// ============================================================
// ADD TO GVL - HMI ROBOT B
// Các biến này mirror trực tiếp biến HMI Robot A.
// AB_StepBlockClipboard / AB_StepCopyCount vẫn dùng chung để có thể copy block step.
// ============================================================
VAR_GLOBAL
    B_PointClipboardName : STRING(20);
    B_PointClipboardR : REAL;
    B_PointClipboardSourceNo : INT;
    B_PointClipboardValid : BOOL;
    B_PointClipboardX : REAL;
    B_PointClipboardY : REAL;
    B_PointClipboardZ : REAL;
    B_StepClipboard : ST_RobotStep;
    B_StepClipboardValid : BOOL;
    B_StepCopyEnd : INT;
    B_StepCopyStart : INT;
    HMI_B_ChangeSelectedPoint : BOOL;
    HMI_B_CondCmdReq : INT;
    HMI_B_CondCmd_Down : BOOL;
    HMI_B_CondCmd_GoBot : BOOL;
    HMI_B_CondCmd_GoTop : BOOL;
    HMI_B_CondCmd_PageDown : BOOL;
    HMI_B_CondCmd_PageUp : BOOL;
    HMI_B_CondCmd_Up : BOOL;
    HMI_B_CondCopied : ST_Condition;
    HMI_B_CondEditEnable : BOOL;
    HMI_B_CondEditIndex : ARRAY[0..10] OF INT;
    HMI_B_CondEditLinkNext : ARRAY[0..10] OF INT;
    HMI_B_CondEditName : STRING(20);
    HMI_B_CondEditNo : INT;
    HMI_B_CondEditNote : ARRAY[0..10] OF STRING(30);
    HMI_B_CondEditOperator : ARRAY[0..10] OF INT;
    HMI_B_CondEditRowEnable : ARRAY[0..10] OF BOOL;
    HMI_B_CondEditSetValue : ARRAY[0..10] OF DINT;
    HMI_B_CondEditSource : ARRAY[0..10] OF INT;
    HMI_B_CondMonActualValue : ARRAY[0..10] OF DINT;
    HMI_B_CondMonFinalResult : BOOL;
    HMI_B_CondMonRowResult : ARRAY[0..10] OF BOOL;
    HMI_B_CondMonitorEnable : BOOL;
    HMI_B_CondRowSelect : ARRAY[0..10] OF BOOL;
    HMI_B_CondSelectedCmd : INT;
    HMI_B_CondSelectedNo : INT;
    HMI_B_CondViewEnable : ARRAY[0..10] OF BOOL;
    HMI_B_CondViewName : ARRAY[0..10] OF STRING(20);
    HMI_B_CondViewNo : ARRAY[0..10] OF INT;
    HMI_B_CondViewResult : ARRAY[0..10] OF BOOL;
    HMI_B_CondViewStart : INT;
    HMI_B_CopyEndStep : INT;
    HMI_B_CopyStartStep : INT;
    HMI_B_EditCmd : E_RobotCmd;
    HMI_B_EditCmdReq : INT;
    HMI_B_EditCmdReq_Arr : ARRAY[0..20] OF BOOL;
    HMI_B_EditGroupCmd : INT;
    HMI_B_EditNote : STRING(20);
    HMI_B_EditP1 : INT;
    HMI_B_EditP2 : INT;
    HMI_B_EditP3 : DINT;
    HMI_B_EditP4 : INT;
    HMI_B_EditP5 : INT;
    HMI_B_EditPointReq : INT;
    HMI_B_EditPointReq_Arr : ARRAY[0..10] OF BOOL;
    HMI_B_EditSelgroupCmd : ARRAY[0..10] OF BOOL;
    HMI_B_EditStepNo : INT;
    HMI_B_Edit_PointNo : INT;
    HMI_B_Edit_Pos_Name : STRING(20);
    HMI_B_Edit_Pos_R : REAL;
    HMI_B_Edit_Pos_X : REAL;
    HMI_B_Edit_Pos_Y : REAL;
    HMI_B_Edit_Pos_Z : REAL;
    HMI_B_Edit_Trigger_Windown_Cmd : ARRAY[0..10] OF BOOL;
    HMI_B_PointNo : ARRAY[0..10] OF INT;
    HMI_B_PointNoSelected : INT;
    HMI_B_PointViewCmd : INT;
    HMI_B_RowSelect : ARRAY[0..10] OF BOOL;
    HMI_B_RowSelectedCmd : INT;
    HMI_B_RowSelectedPoint : INT;
    HMI_B_RowSelectedPoint_Array : ARRAY[0..10] OF BOOL;
    HMI_B_SelectedStepNo : INT;
    HMI_B_ViewCmd : ARRAY[0..10] OF INT;
    HMI_B_ViewCmd_Go_Bot : BOOL;
    HMI_B_ViewCmd_Go_Bot_Old : BOOL;
    HMI_B_ViewCmd_Go_Top : BOOL;
    HMI_B_ViewCmd_Go_Top_Old : BOOL;
    HMI_B_ViewCmd_Page_Down : BOOL;
    HMI_B_ViewCmd_Page_Down_Old : BOOL;
    HMI_B_ViewCmd_Page_Up : BOOL;
    HMI_B_ViewCmd_Page_Up_Old : BOOL;
    HMI_B_ViewCmd_Scroll_Down : BOOL;
    HMI_B_ViewCmd_Scroll_Down_Old : BOOL;
    HMI_B_ViewCmd_Scroll_Up : BOOL;
    HMI_B_ViewCmd_Scroll_Up_Old : BOOL;
    HMI_B_ViewGroupCmd : ARRAY[0..10] OF INT;
    HMI_B_ViewNote : ARRAY[0..10] OF STRING(20);
    HMI_B_ViewP1 : ARRAY[0..10] OF INT;
    HMI_B_ViewP2 : ARRAY[0..10] OF INT;
    HMI_B_ViewP3 : ARRAY[0..10] OF DINT;
    HMI_B_ViewP4 : ARRAY[0..10] OF INT;
    HMI_B_ViewP5 : ARRAY[0..10] OF INT;
    HMI_B_ViewP6 : ARRAY[0..10] OF INT;
    HMI_B_ViewStartPoint : INT;
    HMI_B_ViewStartStep : INT := 1;
    HMI_B_ViewStepNo : ARRAY[0..10] OF INT;
    HMI_B_View_Pos_Name : ARRAY[0..10] OF STRING(20);
    HMI_B_View_Pos_R : ARRAY[0..10] OF REAL;
    HMI_B_View_Pos_X : ARRAY[0..10] OF REAL;
    HMI_B_View_Pos_Y : ARRAY[0..10] OF REAL;
    HMI_B_View_Pos_Z : ARRAY[0..10] OF REAL;
END_VAR

//=============================================================================
// GVL: LOGICAL IO - ROBOT B
//-----------------------------------------------------------------------------
// IO vật lý nên được Map vào các mảng này tại một chương trình riêng.
//=============================================================================
VAR_GLOBAL

    // Command và Status của lệnh TRACK_ON.
	g_stMultiTrackCommandB : ST_MultiToolTrackingCommand;
	g_stMultiTrackStatusB : ST_MultiToolTrackingStatus;
	
	// Cấu hình và Runtime Tool Robot A.
	g_aToolConfigB : ARRAY[0..C_MAX_TOOLS] OF ST_ToolConfig;
	g_aToolStatusB : ARRAY[0..C_MAX_TOOLS] OF ST_ToolStatus;
	
	// Recipe và Queue Robot A.
	g_aMultiTrackRecipeB : ARRAY[0..C_MAX_TRACK_RECIPES] OF ST_MultiToolTrackingRecipe;
	g_stTrackingObjectQueueB : ST_TrackingObjectQueue;
	
	// Cấu hình các nguồn Sensor.
    g_aSensorSourceConfigB : ARRAY[0..C_MAX_SENSOR_SOURCES] OF ST_SensorObjectSourceConfig;

  	// Cấu hình Vision Tracking cho từng Camera/Channel.
	g_aVisionTrackingSourceConfigB : ARRAY[0..C_MAX_VISION_CHANNELS] OF ST_VisionTrackingSourceConfig;
	
	// Multi-object result dành riêng cho Conveyor Tracking.
	g_aVisionTrackingMultiResultB : ARRAY[0..C_MAX_VISION_CHANNELS] OF ST_VisionTrackingMultiResult;
	
	g_aVisionAlignRecipeB : ARRAY[0..C_MAX_VISION_ALIGN_RECIPES] OF ST_VisionAlignRecipe;
	g_aVisionAlignRuntimeB : ARRAY[1..C_MAX_TOOLS] OF ST_VisionAlignToolRuntime;
	g_aTrayConfigB : ARRAY[0..C_MAX_TRAYS] OF ST_TrayConfig;
	g_aTrayRuntimeB : ARRAY[0..C_MAX_TRAYS] OF ST_TrayRuntime;

	
	// Giao tiếp giữa MultiTool Controller và Tracking Core hiện tại.
	g_xMultiTrackCoreExecuteB : BOOL;
	g_xMultiTrackCoreResetB : BOOL;
	g_xMultiTrackCoreAbortB : BOOL;
	g_xMultiTrackPickerSafeB : BOOL;
	
	g_uiMultiTrackObjectIndexB : UINT;
	g_uiMultiTrackToolIDB : UINT;
	g_stMultiTrackPickOffsetB : ST_POS;
	g_rMultiTrackApproachHeightB : REAL;
	
	// Phản hồi từ Tracking Core về MultiTool Controller.
	g_xTrackingCoreAcceptedB : BOOL;
	g_xTrackingCoreBusyB : BOOL;
	g_xTrackingCoreSyncOKB : BOOL;
	g_xTrackingCorePCSInUseB : BOOL;
	g_xTrackingCoreReleasedB : BOOL;
	g_xTrackingCoreErrorB : BOOL;
	g_udiTrackingCoreErrorIDB : UDINT;
	
	// Command Tool được Controller phát ra.
	g_stToolCommandB : ST_ToolCommand;
	
	// Chọn Tool/TCP Robot B.
	g_xSelectToolExecuteB : BOOL;
	g_uiSelectToolIDB : UINT;
	g_stSelectToolTCPB : ST_POS;
	g_xSelectToolDoneB : BOOL;
	g_xSelectToolErrorB : BOOL;
	g_udiSelectToolErrorIDB : UDINT;
	
	// IO logic Tool Robot B.
	// Nếu project đã có mảng IO chung thì dùng mảng cũ và không khai báo lại.
	g_axDIB : ARRAY[0..C_MAX_DI] OF BOOL;
	g_axDORequestToolB : ARRAY[0..C_MAX_DO] OF BOOL;
	
	// Bit test commissioning. Không dùng trong Interpreter chính thức.
	g_xMultiTrackStartTestB : BOOL;
	g_xMultiTrackResetTestB : BOOL;
	g_xMultiTrackAbortTestB : BOOL;
	g_xCreateTestTrackingObjectB : BOOL;
	
	// TRUE khi cấu hình Multi-tool Robot B đã được khởi tạo.
	g_xMultiToolConfigInitializedB : BOOL := FALSE;
	
	// Bit cho phép khởi tạo lại giá trị mặc định khi commissioning.
	g_xInitializeMultiToolConfigB : BOOL := FALSE;
	
	g_xClearTrackingQueueB : BOOL;
	g_xResetTrackingObjectSourceB : BOOL;
	
	//=============================================================================
	// TRACKING APPLICATION RESULT - ROBOT B
	//=============================================================================
	g_xTrackOKB : BOOL;              // TRUE khi lệnh Tracking gần nhất Pick đủ số lượng.
	g_xTrackErrorB : BOOL;           // TRUE khi lệnh Tracking kết thúc lỗi.
	g_udiTrackErrorIDB : UDINT;      // ErrorID của lệnh Tracking gần nhất.
	g_udiTrackDoneCommandIDB : UDINT;// CommandID đã hoàn thành.
	//=============================================================================
	// TOOL COMMAND TỪ INTERPRETER - ROBOT B
	//=============================================================================
	g_stInterpreterToolCommandB : ST_ToolCommand;
	
	g_HMI_PulsePerCycle_Cr_B: REAL;
	g_HMI_PulsePerCycle_Set_B : INT;
	
	// Cho phép test Background Vision Trigger mà chưa cần chạy TRACK_PICK.
	// Production bình thường phải để FALSE.
	g_xVisionTrackingAutoTriggerTestB : BOOL := FALSE;

END_VAR

VAR_GLOBAL
	//=========================================================================

    // VISION REQUEST FROM ROBOT INTERPRETERS

    //=========================================================================

    g_stVisionAlignRequestA : ST_VISION_ALIGN_REQUEST; // Request Vision Align từ Robot A.

    g_stVisionAlignRequestB : ST_VISION_ALIGN_REQUEST; // Request Vision Align từ Robot B.
	
END_VAR

VAR_GLOBAL
	//=============================================================================
	// V5 - CHỈ BỔ SUNG CHO ROBOT B. ROBOT A GIỮ NGUYÊN.
	// Robot A tiếp tục dùng toàn bộ biến generic hiện tại:
	// g_xTrackingMotionAccepted, g_xTrackingMotionBusy, g_xTrackingMotionDone,
	// g_xTrackingMotionError, g_udiTrackingMotionErrorID, g_xTrackingMotionAbortDone,
	// g_xTrackingVacuumOutput, g_xTrackingBlowOutput.
	//=============================================================================
	
	// Tracking state riêng Robot B.
	g_stTrackingConfig_B : ST_TRACKING_CONFIG; // Cấu hình Tracking Robot B.
	g_stTrackingQueue_B : ST_TRACKING_QUEUE; // Queue Object Robot B.
	g_stTrackingRuntime_B : ST_TRACKING_RUNTIME; // Runtime Tracking Robot B.
	
	// Motion handshake riêng Robot B.
	g_xTrackingMotionAcceptedB : BOOL; // Motion Adapter B đã nhận request.
	g_xTrackingMotionBusyB : BOOL; // Motion Tracking B đang chạy.
	g_xTrackingMotionDoneB : BOOL; // Motion Tracking B hoàn thành.
	g_xTrackingMotionErrorB : BOOL; // Motion Tracking B lỗi.
	g_udiTrackingMotionErrorIDB : UDINT; // ErrorID Motion Tracking B.
	g_xTrackingMotionAbortDoneB : BOOL; // Motion B đã Abort xong.
	
	// Debug/output riêng Robot B.
	g_xTrackingVacuumOutputB : BOOL; // VacuumCommand của Tracking Manager B.
	g_xTrackingBlowOutputB : BOOL; // BlowCommand của Tracking Manager B.
	
	// Apply Tool/TCP riêng Robot B.
	g_udiRobotBToolApplyRequestB : UDINT; // RequestID đổi Tool/TCP B.
	g_udiRobotBToolAppliedRequestB : UDINT; // RequestID B đã Apply thành công.
	g_xRobotBToolApplyBusy : BOOL; // B đang Apply Tool/TCP.
	g_xRobotBToolApplyDone : BOOL; // Xung Done Apply Tool/TCP B.
	g_xRobotBToolApplyError : BOOL; // Lỗi Apply Tool/TCP B.
	g_udiRobotBToolApplyErrorID : UDINT; // ErrorID Apply Tool/TCP B.


END_VAR

VAR_GLOBAL
	//=============================================================================
	// HMI TRACKING CONFIG - ROBOT B
	// Chỉ thêm các biến B còn thiếu. Tool Editor B đã tồn tại trong project (4).
	//=============================================================================
	
	// Sensor Source B.
	g_uiHMISensorSourceIndexB : UINT := 1;
	g_stHMISensorSourceB : ST_SensorObjectSourceConfig;
	g_xHMILoadSensorSourceB : BOOL;
	g_xHMISaveSensorSourceB : BOOL;
	g_xHMILoadSensorSourceB_All : BOOL;
	g_xHMISaveSensorSourceB_All : BOOL;
	
	// Tracking Recipe B.
	g_uiHMITrackingRecipeIndexB : UINT := 1;
	g_stHMITrackingRecipeB : ST_MultiToolTrackingRecipe;
	g_xHMILoadTrackingRecipeB : BOOL;
	g_xHMISaveTrackingRecipeB : BOOL;
	g_xHMILoadTrackingRecipeB_All : BOOL;
	g_xHMISaveTrackingRecipeB_All : BOOL;
	
	// Vision Tracking Source B.
	g_uiHMIVisionSourceIndexB : UINT := 1;
	g_stHMIVisionSourceB : ST_VisionTrackingSourceConfig;
	g_xHMILoadVisionSourceB : BOOL;
	g_xHMISaveVisionSourceB : BOOL;
	g_xHMISaveAllVisionSourceB : BOOL;
	g_xHMILoadAllVisionSourceB : BOOL := FALSE;
	
	// Tracking Config B persistence.
	g_xHMITrackingConfigSaveB : BOOL;
	g_xHMITrackingConfigReadB : BOOL;
	
	// Tool Config B persistence.
	// Không dùng g_stHMITool_Config_Save_All của A vì flag hiện tại đang Save g_aToolConfigA.
	g_xHMIToolConfigSaveAllB : BOOL;
	g_xHMIToolConfigReadAllB : BOOL;
	
	//=============================================================================
	// ROBOT B - LAST VISION ALIGN RESULT
	//=============================================================================
	B_VisionHeaderOK : BOOL;                    // Header của Result cuối hợp lệ.
	B_VisionTriggerID : UDINT;                  // TriggerID cuối cùng.
	
	B_VisionX : REAL;                           // X Vision trả về.
	B_VisionY : REAL;                           // Y Vision trả về.
	B_VisionZ : REAL;                           // Z Vision trả về.
	B_VisionA : REAL;                           // Góc Vision trả về.
	B_VisionScore : REAL;                       // Score Vision.
	
END_VAR

// Just_Motion_Control_x86_64_Linux_SM_WV/Application/PRG_ROBOT/POU_MOTION
PROGRAM POU_MOTION
VAR
	// chạy điểm
	MOVP_A :MC_MoveDirectAbsolute;
	MOVP_B :MC_MoveDirectAbsolute;
	// chạy đường thẳng
	MOVL_A: MC_MoveLinearAbsolute;
	MOVL_B: MC_MoveLinearAbsolute;
	// chạy đường tròn
	MOVC_A: MC_MoveCircularAbsolute;
	MOVC_B: MC_MoveCircularAbsolute;
	
	// Biến chạy
	RBA_BufferMode, TestA_BF_Mode: SM3_Robotics.MC_BUFFER_MODE;
	RBA_TransitionMode, TestA_Trans_Mode: SM3_Robotics.MC_TRANSITION_MODE;
	RBA_TransitionParameter, TestA_Tran_Para: ARRAY [0..(SMC_RCNST.MAX_TRANS_PARAMS - 1)] OF LREAL := [500, 0.0];
	RBA_OrientationMode, TestA_Orient_Mode: SM3_Robotics.SMC_ORIENTATION_MODE;
	RBB_BufferMode: SM3_Robotics.MC_BUFFER_MODE;
	RBB_TransitionMode: SM3_Robotics.MC_TRANSITION_MODE;
	RBB_TransitionParameter: ARRAY [0..(SMC_RCNST.MAX_TRANS_PARAMS - 1)] OF LREAL := [500, 0.0] ;
	RBB_OrientationMode: SM3_Robotics.SMC_ORIENTATION_MODE;	
	
	//RBA_MovementType: SM3_Robotics.SMC_PTP_MOVEMENT_TYPE;
	//RBb_MovementType: SM3_Robotics.SMC_PTP_MOVEMENT_TYPE;
	
	Pos_run_manual_A, Pos_run_auto_A , Pos_run_manual_B, Pos_run_auto_B ,
	Pos_Run_A, Pos_Run_A_Pre, Pos_Run_B, Pos_Run_B_Pre : SM3_Robotics.SMC_POS_REF;
	Pos_0 : SM3_Robotics.SMC_POS_REF := (c := (X:= 0,Y:= 0, Z:= 0, A:= 0, B:= 0, C:= 0));	
	MOVL_A_2: MC_MoveLinearAbsolute;
	MOVL_A_3: MC_MoveLinearAbsolute;
	MOVL_B_2: MC_MoveLinearAbsolute;
	MOVL_B_3: MC_MoveLinearAbsolute;
END_VAR

VAR // Act_go_Manual
	Excute_Run_goHome_A , AP_Man_Z_Wait_Go, AP_Man_R_Wait_Go, AP_Man_XY_Wait_Go,
	Excute_Run_goHome_B, Excute_Run_goZ_Wait_B, Excute_Run_goR_Wait_B,Excute_Run_goXY_Wait_B : BOOL;
	AP_Man_Pos_Go , Excute_Run_goPos_A_UpZ, excute_run_L_Upz_A , AP_Man_UP_Z_Go, AP_Man_Pos_Go_L,
 	Excute_Run_goPos_B, Excute_Run_goPos_B_UpZ, excute_run_L_Upz_B , excute_run_P_Upz_B, Excute_Run_goPos_B_L : BOOL;
	Excute_Run_goPos_A_UpZ_XY_BF_R, Excute_Run_goPos_A_UpZ_R_BF_XY, Excute_Run_goPos_B_UpZ_XY_BF_R, Excute_Run_goPos_B_UpZ_R_BF_XY : BOOL;
	excute_run_cam_B, excute_run_cam_A, excute_run_P_cam_B, excute_run_P_cam_A, run_calib_P_Cam_A, run_calib_P_Cam_B : BOOL;
	mode_Run_GoPosA_manual, mode_Run_GoPosB_manual: INT := 0;
	Pro_B_cam : INT;
	Running_B_Cam : BOOL;
	
	
	Other_PosA, Other_PosB: BOOL;
	PRO_A : ARRAY[0..50] OF INT;
	RuningPosA : ARRAY[0..50] OF BOOL;
	PRO_B : ARRAY[0..50] OF INT;
	RuningPosB : ARRAY[0..50] OF BOOL;
	
	T_MC1_4, T_MC2_4, Project_4_Delay_B, Project_4_Delay_A, on_Cam : TON;	
	Project_4_Delay_B1, Project_4_Delay_B2, Project_4_Delay_B3, Project_4_Delay_B4, ton_centering,  
	Project_4_Delay_A1, Project_4_Delay_A2, Project_4_Delay_A3, Project_4_Delay_A4, Project_4_Delay_A5, Project_4_Delay_A6, Project_4_Delay_A7, Project_4_Delay_A8  : TON;
	Ton_OK_MC1_4, Ton_OK_MC2_4, Ton_Limit_Test_TS, Ton_Limit_Test_VS : TON;
	Ton_tacktime, T_Delay_RB_A_Tool_1, T_Delay_RB_A_Tool_2, T_Delay_RB_B_Tool_1, T_Delay_RB_B_Tool_2 : TON;
	on_centering : WORD;
	change_fac_vel_A, change_fac_vel_B : BOOL := FALSE;
	change_fac_vel_max_A, change_fac_vel_max_A_test : BOOL := FALSE;
	change_fac_vel_max_B : BOOL := FALSE;
END_VAR

VAR // Act_go_Auto
	LOG_, LOG_A, LOG_B : FB_Write_Log(); // log file
	i_log, i_log_BF, i_log_HMI : INT;
	{region "1.Project 1"}
		Pallets_get_A,Pallets_put_A,			 
		Pallets_get_B, Pallets_put_B : FB_PALLETS;
			 
		status_MC :INT;	 
			 
		Process_1_A,Process_1_B,
		Process_2_A,Process_2_B: INT;
		Process_2_A_to_B , Process_2_B_to_A : 	 BOOL;
			 
		Process_2_A_1, Process_2_A_2, Process_2_A_3, Process_2_A_4 , 
		Process_2_B_1, Process_2_B_2, Process_2_B_3, Process_2_B_4 : BOOL;

	 
		Blink_Stop, Blink_Start : Blink_Bit; // nháy 
			 
		SR_MC : SR;
		RUN_PROJECT : BOOL;
		INIT_RUN_PROJECT : BOOL;
		AP_Auto_Pos_Go , EXCUTE_RUN_P_AUTO_B , EXCUTE_RUN_L_AUTO_A , EXCUTE_RUN_L_AUTO_B : BOOL;
			 
		Project_2_Delay, Project_2_Delay2 : TON;	  
		
		pr2_mode_A_Pick_to_B_Pick, pr2_mode_A_Pick_to_B_Place : BOOL;			 
		Move_RB_A, Move_RB_B : FB_Run_Point;
		Move_Point_Para_A, Move_Point_Para_B : Move_Point;
	{endregion}
		 
	{region "3.Project 3"}	
 
	Process_3_A,Process_3_B: INT;
	Test_Pick, Test_Place : INT;	 
	run_P_cam_B_test_pick, run_P_cam_B_test_place	: BOOL;	  
		 
	Project_3_Delay_A, Project_3_Delay_B  : TON ;
		 
	A3_Run_P, A3_Run_L, B3_Run_P, B3_Run_L : BOOL;	
	

	A_Comp, B_Comp ,Ena3, B_Allow_NextStep, A_Allow_NextStep, A_Comp_Man, B_Comp_Man, A_FB_Comp, B_FB_Comp, A_Ready, B_Ready : BOOL;
	Pro_A3, Pro_B3 : WORD; 
		  
	nextstepRtrigB, nextstepRtrigA : R_TRIG;
	// Trigger_Cmd, Trigger_Busy, Trigger_Done : BOOL;
	T1_A, T2_A : WORD;
	
	
	DATA_A_T1 , DATA_B_T1, DATA_B_T2 : WORD := 0; // 0 : NONE, 1:barcode // 2 OK 	 // 3 NG 
	DATA_MC1, Data_MC2 : WORD; // 0 NONE, 1 BUSY, 2 ALLOW PLACE, 3 ALLOW PICK 
	ALLOW_PICK_CNV, ALLOW_PLACE_CNV_OK, ALLOW_PLACE_CNV_NG_TS, ALLOW_PLACE_CNV_NG_VS  : BOOL := true;
	Pro_MC1, Pro_MC2 : WORD := 0;
	PRO_A3_,PRO_B3_  : ARRAY[0..10] OF WORD;
		 
	Wait_A3_Run , Pick_A3_Run, Place_A3_Run, Barcode_A3_Run : BOOL := FALSE;	
	 Wait_A3_Finish , Pick_A3_Finish, Place_A3_Finish, Barcode_A3_Finish : BOOL := FALSE;	
 	Allow_MC1, Allow_MC2 : BOOL;
	T_MC1, T_MC2 : TON;	 
	Wait_B3_Run , Pick_B3_T1_Run, Place_OK_B3_T1_Run, Place_NG_B3_T1_Run , Pick_B3_T2_Run , Place_Ok_B3_T2_Run , Place_NG_B3_T2_Run, Barcode_B3_Run: BOOL := FALSE;
	 Wait_B3_Finish , Pick_B3_T1_Finish, Place_OK_B3_T1_Finish, Place_NG_B3_T1_Finish , Pick_B3_T2_Finish , Place_Ok_B3_T2_Finish , Place_NG_B3_T2_Finish , Barcode_B3_Finish : BOOL := FALSE;		   
	{endregion}
    {region "4.Project 4"}
	Pro_B4, Pro_A4, Pro_A4_BF, Pro_B4_BF : WORD; 
	Ena4, Ena_Test : BOOL;	  
	nextstepRtrigB_4, nextstepRtrigA_4 : R_TRIG;
	Trigger_Cmd_4, Trigger_Busy_4, Trigger_Done_4 : BOOL;
	T1_A_4, T2_A_4 : WORD;
	R_Trig_TriggerDone_4 : R_TRIG;
	
	A4_Run_P, A4_Run_L, B4_Run_P, B4_Run_L : BOOL;	
		 
	//GVL.Pro4_.Process.DATA_TOOL_B1_IN , GVL.Pro4_.Process.DATA_TOOL_A1_IN, GVL.Pro4_.Process.DATA_TOOL_A2_OUT, GVL.Pro4_.Process.DATA_TOOL_A1_IN_OLD  : WORD := 0; // 0 : NONE, 1:barcode // 2 OK 	 // 3 NG // 4 - NG TS
	//GVL.Pro4_.Process.DATA_MC_TS, GVL.Pro4_.Process.DATA_MC_VS : WORD; // 0 NONE, 1 BUSY, 2 ALLOW PLACE, 3 ALLOW PICK OK, 4 ALLOW PICK NG, 5 ALLOW PICK NG TS
	ALLOW_PLACE_CNV_OK_4, ALLOW_PLACE_CNV_NG_TS_4, ALLOW_PLACE_CNV_NG_VS_4  : BOOL := TRUE;
	ALLOW_PICK_CNV_4 : BOOL := FALSE;	 
	Pro_MC1_4, Pro_MC2_4 : WORD := 0;
	PRO_B4_,PRO_A4_  : ARRAY[0..10] OF WORD;
		 
	Wait_B4_Run , Pick_B4_Run, Place_B4_Run, Barcode_B4_Run, Trigger_B4_Run : BOOL := FALSE;	
	 Wait_B4_Finish , Pick_B4_Finish, Place_B4_Finish, Barcode_B4_Finish, Trigger_B4_Finish : BOOL := FALSE;	
 	Allow_MC1_4, Allow_MC2_4 : BOOL;
	Ton_Test_B, Ton_Test_A: TON;	 
	delta_position_cor : REAL; 
		 
	Wait_A4_Run , Pick_A4_T1_Run, Place_OK_A4_T1_Run, Place_NG_A4_T1_Run , Pick_A4_T2_Run , Place_Ok_A4_T2_Run , Place_NG_A4_T2_Run, Place_NG_TS_A4_T2_Run, Barcode_A4_Run: BOOL := FALSE;
	 Wait_A4_Finish , Pick_A4_T1_Finish, Place_OK_A4_T1_Finish, Place_NG_A4_T1_Finish , Pick_A4_T2_Finish , Place_Ok_A4_T2_Finish , Place_NG_A4_T2_Finish ,Place_NG_TS_A4_T2_Finish, Barcode_A4_Finish : BOOL := FALSE;
	A_Test_Motion_Run, A_Test_Motion_Finish, B_Test_Motion_Run, B_Test_Motion_Finish, Just_Start_Test : BOOL;
    Process_A_Test, Process_B_Test : WORD;
		 
	D_Barcode_Ts, count_Ts, D_Barcode_Vs, count_Vs, D_Vision_Align_Ts, count_Vs_Align,
	D_CV_NG : WORD;
	T_distance_NG : TON;
	Nb_NG_VS_Cur, Nb_NG_TS_Cur : INT;
	T_Wait_Input_YL, Alarm_Barcode_VS, Alarm_Barcode_TS, Alarm_Full_NG_CONV, T_Wait_Trigger_Bar_TS, T_Wait_Trigger_Bar_VS : TON;
	HeavyAlarm, LightAlarm : BOOL;
	i_Vs_Align, i_Vs_Align_old: INT;
	Process_auto_calib: WORD;
	Run_One_Pos_Calib, Calib_first_bit, NextStep_Test, NextStep_Test_1: BOOL;
	T_Delay_Trigger_Calib: TON;
	Real_to_Word_Pos_Calib : FB_Real_TO_Word_;
	Off_Calib_FtrigB, Off_Calib_FtrigA : F_TRIG;
	Trigger_Calib_Done, Trigger_Auto_Done : R_TRIG;
	Run_Calib_VS_RB : ARRAY[0..GVL.C_MAX_VISION_CHANNELS] OF FB_CalibRunPoints;
	Trigger_VS_FB : ARRAY[0..GVL.C_MAX_VISION_CHANNELS] OF FB_TriggerVS;
	{endregion}
END_VAR

VAR
    step  : ST_RobotStep;
    bCond : BOOL;
END_VAR
//PRG_A_MotionQueueBuilder
VAR
//     step_PRG_A_MotionQueueBuilder : ST_RobotStep;
//     item_PRG_A_MotionQueueBuilder : ST_MotionQueueItem;
//     fbPush : FB_MotionQueuePush;
// 	PushReq : BOOL;
	step_PRG_A_Interpreter : ST_RobotStep;
    fbPushMotion           : FB_MotionQueuePush;
    tRunDelay              : TON;
	WhileReturnStep      : INT;
    MotionCycleResetScan : INT := 0;
END_VAR
// PRG_A_MotionManager
VAR
    fbPop : FB_MotionQueuePop;
	PopReq : BOOL;
    item_PRG_A_MotionManager  : ST_MotionQueueItem;
	freeSlot : INT;
    i : INT;
	fbMoveP : ARRAY[0..3] OF FB_RunMoveP;
    fbMoveL : ARRAY[0..3] OF FB_RunMoveL;
    fbMoveC : ARRAY[0..3] OF FB_RunMoveC;
	SlotPos : ARRAY[0..3] OF SMC_POS_REF;
    SlotMidPos : ARRAY[0..3] OF SMC_POS_REF;
    SlotEndPos : ARRAY[0..3] OF SMC_POS_REF;
	ActiveCountCalc : INT;
	WaitAcceptSlot : INT := 0;
	udiTrackCommandIDA : UDINT; // Id TrackCommand dang thuc hien
	// CommandID của TOOL_RELEASE hiện tại.
	udiToolReleaseCommandIDA : UDINT;
	
	//=============================================================================
	// VISION ALIGN
	//=============================================================================
// 	fbVisionAlignA : FB_VisionAlign;            // FB Vision Align của Robot A.
// 	xVisionAlignStartA : BOOL;                  // Start một chu trình Vision Align.
	uiVisionCameraIDA : UINT := 1;              // Camera của command hiện tại.
	uiVisionJobIDA : UINT := 1;                 // Job của command hiện tại.
	iVisionResultVarA : INT;
	xVisionStepActiveA : BOOL := FALSE;    // THÊM - ownership command Vision riêng Robot A.
	iVisionErrorIDA : INT := 0;    // Lưu ErrorID thực tế của Vision để chẩn đoán lỗi.
END_VAR
VAR
	step_PRG_B_Interpreter : ST_RobotStep;
    fbPushMotion_B           : FB_MotionQueuePush_B;
    tRunDelay_B              : TON;
	WhileReturnStep_B      : INT;
    MotionCycleResetScan_B : INT := 0;
	
	fbPop_B : FB_MotionQueuePop_B;
	PopReq_B : BOOL;
    item_PRG_B_MotionManager  : ST_MotionQueueItem;
	freeSlot_B : INT;
    i_B : INT;
	fbMoveP_B : ARRAY[0..3] OF FB_RunMoveP;
    fbMoveL_B : ARRAY[0..3] OF FB_RunMoveL;
    fbMoveC_B : ARRAY[0..3] OF FB_RunMoveC;
	SlotPos_B : ARRAY[0..3] OF SMC_POS_REF;
    SlotMidPos_B : ARRAY[0..3] OF SMC_POS_REF;
    SlotEndPos_B : ARRAY[0..3] OF SMC_POS_REF;
	ActiveCountCalc_B : INT;
	WaitAcceptSlot_B : INT := 0;
	udiTrackCommandIDB : UDINT; // Id TrackCommand dang thuc hien
	// CommandID của TOOL_RELEASE hiện tại.
	udiToolReleaseCommandIDB : UDINT;
	
	//=============================================================================
	// POU parent localVars - ADD ONLY these missing Robot B Vision interpreter locals.
	// Existing B locals step_PRG_B_Interpreter, fbPushMotion_B, tRunDelay_B,
	// WhileReturnStep_B, MotionCycleResetScan_B, udiTrackCommandIDB and
	// udiToolReleaseCommandIDB already exist in project (4); DO NOT duplicate them.
	//=============================================================================
	uiVisionCameraIDB : UINT := 1;
	uiVisionJobIDB : UINT := 1;
	iVisionResultVarB : INT := 0;
	xVisionStepActiveB : BOOL := FALSE;
	iVisionErrorIDB : INT := 0;
	xVisionAlignStartB : BOOL := FALSE;
	
END_VAR
VAR // added by the converter: edge detectors and wires of the graphical bodies
    _w1, _w2, _w3, _w4, _w5, _w6, _w7 : LREAL;
END_VAR

{region "1.FB Main"}
GVL.Fac_Vel_Slow := 0.03;
// GVL.Fac_Vel_Max_A := 0.4;
// GVL.Fac_Acc_Max_A := 0.4;
// GVL.Fac_Jerk_Max_A := 0.4;	 
// GVL.Fac_Vel_Max_B := 0.4;
// GVL.Fac_Acc_Max_B := 0.4;
// GVL.Fac_Jerk_Max_B := 0.4;
// 	 
// GVL.Fac_Vel_Max_A := GVL_1.DATA_RB_A.Fac_Vel;
// GVL.Fac_Acc_Max_A := GVL_1.DATA_RB_A.Fac_Acc;
// GVL.Fac_Jerk_Max_A := GVL_1.DATA_RB_A.Fac_Jerk;	 
// GVL.Fac_Vel_Max_B := GVL_1.DATA_RB_B.Fac_Vel;
// GVL.Fac_Acc_Max_B := GVL_1.DATA_RB_B.Fac_Acc;
// GVL.Fac_Jerk_Max_B := GVL_1.DATA_RB_B.Fac_Jerk;

	 
IF GVL.RB_A.Auto THEN	 
	IF NOT change_fac_vel_A AND NOT change_fac_vel_max_A_test THEN	 
		GVL.Fac_Vel_Set_A := GVL_1.DATA_RB_A.Fac_Vel;
		GVL.Fac_Acc_Set_A := GVL_1.DATA_RB_A.Fac_Acc;
		GVL.Fac_Jerk_Set_A := GVL_1.DATA_RB_A.Fac_Jerk;
		GVL.Fac_Torque_Set_A := GVL_1.DATA_RB_A.Fac_Torque;
	ELSE
		IF change_fac_vel_A THEN
			GVL.Fac_Vel_Set_A := GVL.Fac_Vel_Slow;
			GVL.Fac_Acc_Set_A := GVL_1.DATA_RB_A.Fac_Acc;
			GVL.Fac_Jerk_Set_A := GVL_1.DATA_RB_A.Fac_Jerk;
			GVL.Fac_Torque_Set_A := GVL_1.DATA_RB_A.Fac_Torque;
		END_IF;
		IF change_fac_vel_max_A_test THEN
			GVL.Fac_Vel_Set_A := GVL.Pro4_.Auto.Fac_Vel_Max_A;	 
			GVL.Fac_Acc_Set_A := GVL.Pro4_.Auto.Fac_Acc_Max_A;
			GVL.Fac_Jerk_Set_A := GVL.Pro4_.Auto.Fac_Jerk_Max_A;
		END_IF;
	END_IF;
ELSE
	GVL.Fac_Vel_Set_A := GVL_1.DATA_RB_A.Fac_Vel_Man;
	GVL.Fac_Acc_Set_A := GVL_1.DATA_RB_A.Fac_Acc_Man;
	GVL.Fac_Jerk_Set_A := GVL_1.DATA_RB_A.Fac_Jerk_Man;
	GVL.Fac_Torque_Set_A := GVL_1.DATA_RB_A.Fac_Torque; 
END_IF

IF GVL.RB_B.Auto THEN		 
	IF NOT change_fac_vel_B AND NOT change_fac_vel_max_B THEN	 
		GVL.Fac_Vel_Set_B := GVL_1.DATA_RB_B.Fac_Vel;
		GVL.Fac_Acc_Set_B := GVL_1.DATA_RB_B.Fac_Acc;
		GVL.Fac_Jerk_Set_B := GVL_1.DATA_RB_B.Fac_Jerk;
		GVL.Fac_Torque_Set_B := GVL_1.DATA_RB_B.Fac_Torque;
	ELSE
		IF change_fac_vel_B THEN
			GVL.Fac_Vel_Set_B := GVL.Fac_Vel_Slow;
			GVL.Fac_Acc_Set_B := GVL_1.DATA_RB_B.Fac_Acc;
			GVL.Fac_Jerk_Set_B := GVL_1.DATA_RB_B.Fac_Jerk;	
			GVL.Fac_Torque_Set_B := GVL_1.DATA_RB_B.Fac_Torque; 
		END_IF;
		IF change_fac_vel_max_B THEN
			GVL.Fac_Vel_Set_B := GVL.Pro4_.Auto.Fac_Vel_Max_B;	 
			GVL.Fac_Acc_Set_B := GVL.Pro4_.Auto.Fac_Acc_Max_B;
			GVL.Fac_Jerk_Set_B := GVL.Pro4_.Auto.Fac_Jerk_Max_B;
		END_IF
	END_IF
ELSE
	GVL.Fac_Vel_Set_B := GVL_1.DATA_RB_B.Fac_Vel_Man;
	GVL.Fac_Acc_Set_B := GVL_1.DATA_RB_B.Fac_Acc_Man;
	GVL.Fac_Jerk_Set_B := GVL_1.DATA_RB_B.Fac_Jerk_Man;
	GVL.Fac_Torque_Set_B := GVL_1.DATA_RB_B.Fac_Torque_Man;	 
END_IF
	 
// IF NOT change_fac_vel_max_B THEN
// 	GVL.Fac_Vel_Set_B := GVL_1.DATA_RB_B.Fac_Vel;
// 	GVL.Fac_Acc_Set_B := GVL_1.DATA_RB_B.Fac_Acc;
// 	GVL.Fac_Jerk_Set_B := GVL_1.DATA_RB_B.Fac_Jerk;
// ELSE
// 	GVL.Fac_Vel_Set_B := GVL.Pro4_.Auto.Fac_Vel_Max_B;	 
// 	GVL.Fac_Acc_Set_B := GVL.Pro4_.Auto.Fac_Acc_Max_B;
// 	GVL.Fac_Jerk_Set_B := GVL.Pro4_.Auto.Fac_Jerk_Max_B;
// END_IF
	 
//namnv0104
IF GVL.Pro4_.Signal_In.T_Cv_NG_out_full.Q THEN
	GVL.Pro4_.Auto.NG_CV_Full_Pro := TRUE;
ELSE
	GVL.Pro4_.Auto.NG_CV_Full_Pro := FALSE;
END_IF;
M_reset();
MOVC(); MOVL(); 	 	  
MOVP(); 

ACT_Excute_Run(); // Bit Controll
ACT_GO_Pos_Manual(); // set điểm & call
ACT_GO_Pos_Auto(); // Auto

IF GVL.MB_[6] THEN
	GVL.RB_A_.Tool_1 := FALSE;
	GVL.RB_B_.Tool_1 := FALSE;
END_IF;	 
{endregion}
{region "2. PRAMETER"}
/// Tham so
// RBA_BufferMode := 0; 
// RBA_BufferMode := MC_BUFFER_MODE.Aborting; 
RBA_OrientationMode := SM3_Robotics.SMC_ORIENTATION_MODE.Axis; // 0 : axis- 1: cicle
RBA_TransitionMode := SM3_Robotics.MC_TRANSITION_MODE.TMNone;
	 
	 
//RBB_BufferMode := 0;
//RBB_BufferMode := SM3_Robotics.MC_BUFFER_MODE.Aborting; 
RBB_OrientationMode := SM3_Robotics.SMC_ORIENTATION_MODE.Axis;
RBB_TransitionMode := SM3_Robotics.MC_TRANSITION_MODE.TMNone;
	 
{endregion}
{region "3. POS_MAN OR AUTO"}
/// Manual or Auto 1
IF GVL.RB_A.Manual AND NOT GVL.RB_A.Auto THEN
	Pos_Run_A := Pos_run_manual_A;
ELSIF NOT GVL.RB_A.Manual AND GVL.RB_A.Auto THEN
	Pos_Run_A := Pos_run_auto_A;
ELSE
	Pos_Run_A := Pos_0;
END_IF;
/// Manual or Auto 2
IF GVL.RB_B.Manual AND NOT GVL.RB_B.Auto THEN
	Pos_Run_B := Pos_run_manual_B;
ELSIF NOT GVL.RB_b.Manual AND GVL.RB_b.Auto THEN
	Pos_Run_B := Pos_run_auto_B;
ELSE
	Pos_Run_B := Pos_0;
END_IF;
{endregion}
// Log_Machine	 
FOR i_log := 1 TO 20 DO
    // GVL.Log_HMI[i_log] := LOG_.Buffer[i_log];
	GVL.Log_RobotA[i_log] := LOG_A.Buffer[i_log];
	GVL.Log_RobotB[i_log] := LOG_B.Buffer[i_log];
END_FOR
i_log_HMI := 1;
FOR i_log_BF := LOG_.Index TO 1 BY -1 DO
	GVL.Log_HMI[i_log_HMI] := LOG_.Buffer[i_log_BF];
	i_log_HMI := i_log_HMI + 1;
END_FOR

// Thuc hien ham trigger VS Cam ID 0
Trigger_VS_FB[0](Enable := GVL.Auto_VS_RB[0].Enable_FB_Trigger_VS,
				 Start := GVL.Auto_VS_RB[0].Start_FB_Trigger_VS,
				 count_Vs_Align_max := GVL.Data_Calib_RB[0].Nb_Trigger_VS_Max,
				 T_Delay_Trigger_time := GVL.Data_Calib_RB[0].Delay_Trigger_Time,
// 				 Trigger_RB := GVL.Auto_VS_RB[0].Trigger_VS, // Bien trigger robot A gui Vision
// 				 Triger_RB_Done := GVL.Auto_VS_RB[0].Trigger_Done, //Bien trigger done Vision gui robot A
				 Trigger_Again := GVL.Auto_VS_RB[0].Trigger_Again,
				 Pass_Triger_VS_NG := GVL.Auto_VS_RB[0].Pass_Trigger_VS_NG,
				 Mode_ByPass_VS := GVL.Data_Calib_RB[0].Bypass_VS,
	);

ACTION MOVC:
MOVC_B(
    AxisGroup := SCARA_B,
    Velocity := TO_LREAL(GVL.RB_B.SPEED),
    Acceleration := TO_LREAL(GVL.RB_B.ACC),
    Deceleration := TO_LREAL(GVL.RB_B.DEC),
    Jerk := TO_LREAL(GVL.RB_B.JERK),
    CoordSystem := GVL.RB_b.COORD,
    BufferMode := RBB_BufferMode,
    TransitionMode := RBB_TransitionMode,
    TransitionParameter := RBB_TransitionParameter,
    OrientationMode := RBB_OrientationMode,
    VelFactor := TO_LREAL(GVL.Fac_Vel_Set_B),
    AccFactor := TO_LREAL(GVL.Fac_Acc_Set_B),
    JerkFactor := TO_LREAL(GVL.Fac_Jerk_Set_B),
    TorqueFactor := TO_LREAL(GVL.Fac_Torque_Set_B)); // MC_MoveCircularAbsolute
MOVC_A(
    AxisGroup := SCARA_A,
    Velocity := TO_LREAL(GVL.RB_A.SPEED),
    Acceleration := TO_LREAL(GVL.RB_A.ACC),
    Deceleration := TO_LREAL(GVL.RB_A.DEC),
    Jerk := TO_LREAL(GVL.RB_A.JERK),
    CoordSystem := GVL.RB_A.COORD,
    BufferMode := RBA_BufferMode,
    TransitionMode := RBA_TransitionMode,
    TransitionParameter := RBA_TransitionParameter,
    OrientationMode := RBA_OrientationMode,
    VelFactor := TO_LREAL(GVL.Fac_Vel_Set_A),
    AccFactor := TO_LREAL(GVL.Fac_Acc_Set_A),
    JerkFactor := TO_LREAL(GVL.Fac_Jerk_Set_A),
    TorqueFactor := TO_LREAL(GVL.Fac_Torque_Set_A)); // MC_MoveCircularAbsolute
END_ACTION

ACTION MOVL:
_w1 := TO_LREAL(GVL.RB_B.SPEED);
_w2 := TO_LREAL(GVL.RB_B.ACC);
_w3 := TO_LREAL(GVL.RB_B.DEC);
_w4 := TO_LREAL(GVL.RB_B.JERK);
_w5 := TO_LREAL(GVL.Fac_Vel_Set_B);
_w6 := TO_LREAL(GVL.Fac_Acc_Set_B);
_w7 := TO_LREAL(GVL.Fac_Jerk_Set_B);
MOVL_A(
    AxisGroup := SCARA_A,
    Position := Pos_Run_A,
    Velocity := TO_LREAL(GVL.RB_A.SPEED),
    Acceleration := TO_LREAL(GVL.RB_A.ACC),
    Deceleration := TO_LREAL(GVL.RB_A.DEC),
    Jerk := TO_LREAL(GVL.RB_A.JERK),
    CoordSystem := GVL.RB_A.COORD,
    BufferMode := RBA_BufferMode,
    TransitionMode := RBA_TransitionMode,
    TransitionParameter := RBA_TransitionParameter,
    OrientationMode := RBA_OrientationMode,
    VelFactor := TO_LREAL(GVL.Fac_Vel_Set_A),
    AccFactor := TO_LREAL(GVL.Fac_Acc_Set_A),
    JerkFactor := TO_LREAL(GVL.Fac_Jerk_Set_A),
    TorqueFactor := TO_LREAL(GVL.Fac_Torque_Set_A)); // MC_MoveLinearAbsolute
MOVL_B(
    AxisGroup := SCARA_B,
    Position := Pos_Run_B,
    Velocity := _w1,
    Acceleration := _w2,
    Deceleration := _w3,
    Jerk := _w4,
    CoordSystem := GVL.RB_b.COORD,
    BufferMode := RBB_BufferMode,
    TransitionMode := RBB_TransitionMode,
    TransitionParameter := RBB_TransitionParameter,
    OrientationMode := RBB_OrientationMode,
    VelFactor := _w5,
    AccFactor := _w6,
    JerkFactor := _w7,
    TorqueFactor := TO_LREAL(GVL.Fac_Torque_Set_B)); // MC_MoveLinearAbsolute
END_ACTION

ACTION MOVP:
MOVP_A(
    AxisGroup := SCARA_A,
    Position := Pos_Run_A,
    CoordSystem := GVL.RB_A.COORD,
    BufferMode := RBA_BufferMode,
    TransitionMode := RBA_TransitionMode,
    TransitionParameter := RBA_TransitionParameter,
    VelFactor := TO_LREAL(GVL.Fac_Vel_Set_A),
    AccFactor := TO_LREAL(GVL.Fac_Acc_Set_A),
    JerkFactor := TO_LREAL(GVL.Fac_Jerk_Set_A),
    TorqueFactor := TO_LREAL(GVL.Fac_Torque_Set_A)); // MC_MoveDirectAbsolute
MOVP_B(
    AxisGroup := SCARA_B,
    Position := Pos_Run_B,
    CoordSystem := GVL.RB_B.COORD,
    BufferMode := RBB_BufferMode,
    TransitionMode := RBB_TransitionMode,
    TransitionParameter := RBB_TransitionParameter,
    VelFactor := TO_LREAL(GVL.Fac_Vel_Set_B),
    AccFactor := TO_LREAL(GVL.Fac_Acc_Set_B),
    JerkFactor := TO_LREAL(GVL.Fac_Jerk_Set_B),
    TorqueFactor := TO_LREAL(GVL.Fac_Torque_Set_B)); // MC_MoveDirectAbsolute
END_ACTION

ACTION ACT_GO_Pos_Auto:
Blink_Start(Enable	:= TRUE);
Blink_Stop(Enable	:= TRUE);

// M_LoadData(); // pro3
// control lamp
GVL.HMI_MAIN.yLamp_Yellow := T_Wait_Input_YL.Q AND GVL.HMI_MAIN.yStart;
HeavyAlarm := FALSE;
//HeavyAlarm :=  GVL.Alarm_Robot.A_Tool_1 OR GVL.Alarm_Robot.A_Tool_2 OR GVL.Alarm_Robot.B_Tool_1 OR GVL.Alarm_Robot.B_Tool_2;
LightAlarm := GVL.Alarm_P4.Alarm_Limit_NG_TS OR GVL.Alarm_P4.Alarm_Limit_NG_VS OR Alarm_Full_NG_CONV.Q OR Alarm_Barcode_TS.Q OR Alarm_Barcode_VS.Q OR GVL.Alarm_P4.Alarm_Limit_Test_TS OR GVL.Alarm_P4.Alarm_Limit_Test_VS;
GVL.HMI_MAIN.yBuzz := HeavyAlarm OR LightAlarm;

	// AND GVL.RB_B.Auto
SR_MC(	SET1 := GVL.HMI_MAIN.Start AND (GVL.RB_A.Auto OR GVL.RB_B.Auto) ,
		RESET := GVL.HMI_MAIN.Stop OR NOT GVL.X[9] OR GVL.RB_A.Manual OR GVL.RB_B.Manual OR HeavyAlarm,
		Q1 => RUN_PROJECT);	
	  
gVL.HMI_MAIN.yStop := NOT RUN_PROJECT ;
GVL.HMI_MAIN.yStart := RUN_PROJECT ;
delta_position_cor := 0.02;
//GVL.HMI_MAIN.yStart := RUN_PROJECT OR ( NOT Blink_Start.Out AND (GVL.RB_A.Auto OR GVL.RB_B.Auto)) ;
IF (MOVP_A.Done OR MOVL_A.Done) 
AND (ABS(GVL.RB_A_.CUR_X - Pos_run_auto_A.c.X) < delta_position_cor) 
AND (ABS(GVL.RB_A_.CUR_Y - Pos_run_auto_A.c.Y) < delta_position_cor) 
AND (ABS(GVL.RB_A_.CUR_Z - Pos_run_auto_A.c.Z) < delta_position_cor) 
AND (ABS(GVL.RB_A_.CUR_R - Pos_run_auto_A.c.A) < delta_position_cor)
THEN  A_Comp	:= TRUE;  ELSE A_Comp	:= FALSE; END_IF;

IF (MOVP_A.Done OR MOVL_A.Done) THEN  A_FB_Comp := TRUE; ELSE A_FB_Comp	:= FALSE; END_IF;

IF (NOT MOVP_A.Done AND NOT MOVL_A.Done AND NOT MOVP_A.Execute AND NOT MOVL_A.Execute)
AND (ABS(Pos_Run_A.c.X - Pos_run_auto_A.c.X) < delta_position_cor) 
AND (ABS(Pos_Run_A.c.Y - Pos_run_auto_A.c.Y) < delta_position_cor) 
AND (ABS(Pos_Run_A.c.Z - Pos_run_auto_A.c.Z) < delta_position_cor) 
AND (ABS(Pos_Run_A.c.A - Pos_run_auto_A.c.A) < delta_position_cor)
THEN  A_Ready	:= TRUE;  ELSE A_Ready	:= FALSE; END_IF;

IF (MOVP_B.Done OR MOVL_B.Done)  
AND (ABS(GVL.RB_B_.CUR_X - Pos_run_auto_B.c.X) < delta_position_cor) 
AND (ABS(GVL.RB_B_.CUR_Y - Pos_run_auto_B.c.Y) < delta_position_cor) 
AND (ABS(GVL.RB_B_.CUR_Z - Pos_run_auto_B.c.Z) < delta_position_cor) 
AND (ABS(GVL.RB_B_.CUR_R - Pos_run_auto_B.c.A) < delta_position_cor)
THEN  B_Comp	:= TRUE;  ELSE B_Comp	:= FALSE; END_IF;

IF (MOVP_B.Done OR MOVL_B.Done) THEN  B_FB_Comp	:= TRUE; ELSE B_FB_Comp	:= FALSE; END_IF;

IF (NOT MOVP_B.Done AND NOT MOVL_B.Done AND NOT MOVP_B.Execute AND NOT MOVL_B.Execute)
AND (ABS(Pos_Run_B.c.X - Pos_run_auto_B.c.X) < delta_position_cor) 
AND (ABS(Pos_Run_B.c.Y - Pos_run_auto_B.c.Y) < delta_position_cor) 
AND (ABS(Pos_Run_B.c.Z - Pos_run_auto_B.c.Z) < delta_position_cor) 
AND (ABS(Pos_Run_B.c.A - Pos_run_auto_B.c.A) < delta_position_cor)
THEN  B_Ready	:= TRUE;  ELSE B_Ready	:= FALSE; END_IF;
// Cai dat cac tham so khi chay Auto
IF GVL.ProjectAndModel.Direction_Robot_Current = 0 THEN
	Move_Point_Para_A.Hand_Type := 0;
	Move_Point_Para_B.Hand_Type := 1;
ELSE
	Move_Point_Para_A.Hand_Type := 1;
	Move_Point_Para_B.Hand_Type := 0;
END_IF

// Cai dat tham so bao Error 
IF MOVP_A.Error OR MOVL_A.Error THEN
	Move_Point_Para_A.A_Error := TRUE;
	Move_Point_Para_B.A_Error := TRUE;
ELSE
	Move_Point_Para_A.A_Error := FALSE;
	Move_Point_Para_B.A_Error := FALSE;
END_IF

IF MOVP_B.Error OR MOVL_B.Error THEN
	Move_Point_Para_A.B_Error := TRUE;
	Move_Point_Para_B.B_Error := TRUE;
ELSE
	Move_Point_Para_A.B_Error := FALSE;
	Move_Point_Para_B.B_Error := FALSE;
END_IF



IF NOT RUN_PROJECT THEN
	INIT_RUN_PROJECT := FALSE;
	change_fac_vel_A := FALSE;
	change_fac_vel_max_A_test := FALSE;
	change_fac_vel_B := FALSE;
	change_fac_vel_max_B := FALSE;
	//reset trang thai dieu khien RB-A, RB-B
	Move_Point_Para_A.Enable := FALSE;
	Move_Point_Para_B.Enable := FALSE;
END_IF

Move_RB_A(Enable := Move_Point_Para_A.Enable,
			  Hand_Type := Move_Point_Para_A.Hand_Type, 
			  Move_Type := Move_Point_Para_A.Move_Type,
			  A_Error := Move_Point_Para_A.A_Error,
			  B_Error := Move_Point_Para_A.B_Error,
			  A_Ready := A_Ready,
			  B_Ready := B_Ready,
			  A_Comp := A_Comp,
			  B_Comp := B_Comp,
			  ARunP := A4_Run_P,
			  ARunL := A4_Run_L,
			  BRunP := B4_Run_P,
			  BRunL := B4_Run_L
	);
Move_RB_B(Enable := Move_Point_Para_B.Enable,
		  Hand_Type := Move_Point_Para_B.Hand_Type, 
		  Move_Type := Move_Point_Para_B.Move_Type,
		  A_Error := Move_Point_Para_B.A_Error,
		  B_Error := Move_Point_Para_B.B_Error,
		  A_Ready := A_Ready,
		  B_Ready := B_Ready,
		  A_Comp := A_Comp,
		  B_Comp := B_Comp,
		  ARunP := A4_Run_P,
		  ARunL := A4_Run_L,
		  BRunP := B4_Run_P,
		  BRunL := B4_Run_L
	);


	
IF RUN_PROJECT THEN
	LOG_.Write('Machine Auto Run');
	// namnv1405	  
	CASE GVL.ProjectAndModel.Project_No_Current OF
		0:
			LOG_.Write('Run Test No Vission');
			Ena_Test := TRUE;
			_Main_Process_Test();
			//_Main_Process_Test_VS();
		1:
			LOG_.Write('Run Test With Vission');
			//M_Project_1(ena:= TRUE);  // Array Pick & Place
			Ena_Test := TRUE;
			//_Main_Process_Test();
			_Main_Process_Test_VS();
		2:
			LOG_.Write('Run Project 2');
			//M_Project_2(Ena := TRUE);	// Pick & Place RB A - RB B	
		3:
			LOG_.Write('Run Project 3');
			Ena3:= TRUE;
			//_Main_Process();	 // Project align vision Robot B
		4: 
			
			IF NOT INIT_RUN_PROJECT THEN

				LOG_.Write('Run Project 4');
				INIT_RUN_PROJECT := TRUE;
			END_IF

			Ena4:= TRUE;
			_Main_Process_4();	 // Project align vision Robot B
			
	END_CASE	
ELSE
	A_Comp  := FALSE;
	B_Comp	:= FALSE;
	Ena3	:= FALSE;
	Ena4 	:= FALSE;
	Ena_Test := FALSE;
	A_Test_Motion_Run := FALSE;
	B_Test_Motion_Run := FALSE;
	Just_Start_Test := FALSE;
	//_Main_Process();
	//_Main_Process_4();	
	GVL.Auto_VS_RB[0].Enable_FB_Trigger_VS := FALSE;
	GVL.Auto_VS_RB[0].Start_FB_Trigger_VS := FALSE;
END_IF;


/// 
GVL_2.Process3.Pro_A := Pro_A3;
GVL_2.Process3.Pro_B := Pro_B3;

Main_Base_Program_RB_A();
PRG_A_MotionManager();


Main_Base_Program_RB_B();
PRG_B_MotionManager();
END_ACTION

ACTION Main_Base_Program_RB_A:
//====================================================
// PRG_A_Interpreter
// Controlled Pipeline:
// - Motion được nạp trước tối đa A_PipelineDepth lệnh.
// - A_RunStep chỉ tăng khi step hiện tại Done thật.
// - Gặp lệnh logic thì chờ Motion Queue + Slot sạch.
//====================================================



//====================================================
// STOP COMMAND
//====================================================
IF GVL.A_RunStop OR GVL.X[7] THEN

    // Dừng Interpreter
    GVL.A_RunEnable := FALSE;
    GVL.A_RunBusy := FALSE;
    GVL.A_RunDone := FALSE;
    GVL.A_RunPause := FALSE;
    GVL.A_RunState := 0;
    // GVL.A_RunStop := FALSE;

    // Dừng pipeline
    GVL.A_PipelineActive := FALSE;
    GVL.A_PushMotionReq := FALSE;
    GVL.A_PushMotionDone := FALSE;
    GVL.A_PushMotionError := FALSE;
	// 1707
	//------------------------------------------------
    // Reset bộ nhớ cạnh của FB Push
    //------------------------------------------------
    fbPushMotion(
        Execute := FALSE,
        Item := GVL.A_PushMotionItem
    );

    // Yêu cầu MotionManager abort toàn bộ motion pipeline
    GVL.A_MotionAbortReq := TRUE;
	
	// Dừng command Tracking đang chạy.
	IF GVL.A_StepActive THEN
		GVL.g_stMultiTrackCommandA.Abort := TRUE;
		GVL.g_stMultiTrackCommandA.Execute := FALSE;
	
		GVL.A_StepActive := FALSE;
		udiTrackCommandIDA := 0;
	END_IF;
	
	// Hủy Tool command từ Interpreter.
	GVL.g_stInterpreterToolCommandA.Execute := FALSE;
	GVL.g_stInterpreterToolCommandA.Abort := TRUE;
	
	udiToolReleaseCommandIDA := 0;
	// GVL.A_StepActive := FALSE;
	//GVL.g_axDORequestToolA[4] := FALSE;
	
	//xVisionAlignStartA := FALSE;
	// Hủy Vision Request khi Stop/Disable Robot A.

    //=============================================================================
	// ABORT VISION REQUEST - ROBOT A
	//-----------------------------------------------------------------------------
	// Khi Robot Stop, Robot không phát Request mới và hạ Execute hiện tại.
	// Vision Manager sẽ thực hiện phần reset handshake phía Manager.
	//=============================================================================
	GVL.g_stVisionAlignRequestA.Execute := FALSE;
	xVisionStepActiveA := FALSE;

    RETURN;
END_IF;


//====================================================
// NOT ENABLE
//====================================================
IF NOT GVL.A_RunEnable THEN
    GVL.A_RunBusy := FALSE;
    GVL.A_RunState := 0;
    GVL.A_PushMotionReq := FALSE;
    GVL.A_PipelineActive := FALSE;
	GVL.A_RunAlarm := FALSE;
	GVL.A_RunStep := 1;
	
	GVL.g_stMultiTrackCommandA.Execute := FALSE;
	GVL.g_stMultiTrackCommandA.Abort := FALSE;
	GVL.g_stMultiTrackCommandA.Reset := FALSE;
	
	GVL.A_StepActive := FALSE;
	udiTrackCommandIDA := 0;
	
	GVL.g_stInterpreterToolCommandA.Execute := FALSE;
	GVL.g_stInterpreterToolCommandA.Abort := FALSE;
	GVL.g_stInterpreterToolCommandA.Reset := FALSE;
	
	udiToolReleaseCommandIDA := 0;
	
	// Reset command Vision của Interpreter.
	//xVisionAlignStartA := FALSE;
// 	uiVisionCameraIDA := 1;
// 	uiVisionJobIDA := 1;

	// Hủy Vision Request khi Stop/Disable Robot A.

    GVL.g_stVisionAlignRequestA.Execute := FALSE;   // Hạ Request để Manager kết thúc handshake.

    xVisionStepActiveA := FALSE;                    // Xóa ownership command Vision Robot A.

    uiVisionCameraIDA := 1;                         // Reset CameraID mặc định nếu cần.

    uiVisionJobIDA := 1;                            // Reset JobID mặc định nếu cần.

    iVisionResultVarA := 0;                         // Reset index biến kết quả.
	
	GVL.A_VisionDone := FALSE;
	GVL.A_VisionOK := FALSE;
	GVL.A_VisionError := FALSE;

    RETURN;
END_IF;


//====================================================
// PAUSE
// Pause chỉ dừng Interpreter, không reset Motion đang chạy
//====================================================
IF GVL.A_RunPause THEN
    GVL.A_RunBusy := TRUE;
    RETURN;
END_IF;


//====================================================
// ALARM
//====================================================
IF GVL.A_RunAlarm THEN
    GVL.A_RunBusy := FALSE;
    GVL.A_PushMotionReq := FALSE;
    GVL.A_PipelineActive := FALSE;

    // Khi lỗi thì yêu cầu MotionManager ngừng cấp lệnh mới
    GVL.A_MotionAbortReq := TRUE;

    RETURN;
END_IF;


//====================================================
// RUNNING
//====================================================
GVL.A_RunBusy := TRUE;


//====================================================
// CHECK STEP RANGE
//====================================================
IF GVL.A_RunStep < 1 THEN
    GVL.A_RunStep := 1;
END_IF;

IF GVL.A_RunStep > GVL.A_LengthStep THEN
    GVL.A_RunEnable := FALSE;
    GVL.A_RunBusy := FALSE;
    GVL.A_RunDone := TRUE;
    GVL.A_RunState := 0;
    GVL.A_PipelineActive := FALSE;
    GVL.A_PushMotionReq := FALSE;
	GVL.A_RunStep := 1;
    RETURN;
END_IF;


//====================================================
// STEP RUN EDGE
// Bắt xung nút chạy từng bước từ HMI
//====================================================
GVL.A_StepRunEdge := GVL.A_StepRunReq AND NOT GVL.A_LastStepRunReq;
GVL.A_LastStepRunReq := GVL.A_StepRunReq;


//====================================================
// STEP HOLD
// Nếu đang ở chế độ Step và đang Hold
// thì chỉ chạy tiếp khi có xung StepRun
//====================================================
IF GVL.A_RunMode = 1 THEN

    IF GVL.A_StepHold THEN

        IF GVL.A_StepRunEdge THEN
            // Cho phép chạy 1 step tiếp theo
            GVL.A_StepHold := FALSE;
        ELSE
            // Chưa bấm Step thì đứng yên
            GVL.A_RunBusy := TRUE;
            RETURN;
        END_IF;

    END_IF;

END_IF;


CASE GVL.A_RunState OF

    0: // READ STEP

        step_PRG_A_Interpreter := GVL_1.Step_Cr_A[GVL.A_RunStep];

        IF F_IsMotionCmd(step_PRG_A_Interpreter.Cmd) THEN

            // Bắt đầu pipeline tại step hiện tại
            GVL.A_PipelineActive := TRUE;

            // Step tiếp theo cần push vào motion queue
            GVL.A_PipelineNextPushStep := GVL.A_RunStep;

            GVL.A_RunState := 100;

        ELSE

            // Lệnh logic chỉ được chạy khi toàn bộ motion đã sạch
            IF (GVL.A_MotionCount <= 0) AND (GVL.A_ActiveMotionCount <= 0) THEN
                GVL.A_RunState := 10;
            ELSE
                GVL.A_RunState := 130;
            END_IF;

        END_IF;


    10: // EXECUTE LOGIC COMMAND

        step_PRG_A_Interpreter := GVL_1.Step_Cr_A[GVL.A_RunStep];

        CASE step_PRG_A_Interpreter.Cmd OF

            E_RobotCmd.CMD_NOP:
                GVL.A_RunStep := GVL.A_RunStep + 1;
                GVL.A_RunState := 0;


            E_RobotCmd.CMD_Set_Speed:
                // P1 = Speed, P2 = Acc, P3 = Dec, P4 = Jerk
                GVL.A_CurrentMotionParam.Speed := INT_TO_LREAL(step_PRG_A_Interpreter.P1);
                GVL_1.DATA_RB_A.MOTION_ACC  := INT_TO_LREAL(step_PRG_A_Interpreter.P2);
                GVL_1.DATA_RB_A.MOTION_DEC  := DINT_TO_LREAL(step_PRG_A_Interpreter.P3);
                GVL_1.DATA_RB_A.MOTION_JERK := INT_TO_LREAL(step_PRG_A_Interpreter.P4);

                GVL.A_RunStep := GVL.A_RunStep + 1;
                GVL.A_RunState := 0;
				// Nếu đang Step Mode thì dừng chờ sau khi chạy xong 1 lệnh
				IF GVL.A_RunMode = 1 THEN
					GVL.A_StepHold := TRUE;
				END_IF;

            E_RobotCmd.CMD_Set_Fac_Speed:
                // P1 = VelFac %, P2 = AccFac %, P4 = JerkFac %
                GVL_1.DATA_RB_A.Fac_Vel  := INT_TO_LREAL(step_PRG_A_Interpreter.P1) / 100.0;
                GVL_1.DATA_RB_A.Fac_Acc  := INT_TO_LREAL(step_PRG_A_Interpreter.P2) / 100.0;
                GVL_1.DATA_RB_A.Fac_Jerk := INT_TO_LREAL(step_PRG_A_Interpreter.P4) / 100.0;

                IF GVL_1.DATA_RB_A.Fac_Vel <= 0.0 THEN GVL_1.DATA_RB_A.Fac_Vel := 0.1; END_IF;
                IF GVL_1.DATA_RB_A.Fac_Acc <= 0.0 THEN GVL_1.DATA_RB_A.Fac_Acc := 0.1; END_IF;
                IF GVL_1.DATA_RB_A.Fac_Jerk <= 0.0 THEN GVL_1.DATA_RB_A.Fac_Jerk := 0.1; END_IF;

                GVL.A_RunStep := GVL.A_RunStep + 1;
                GVL.A_RunState := 0;
				
				// Nếu đang Step Mode thì dừng chờ sau khi chạy xong 1 lệnh
				IF GVL.A_RunMode = 1 THEN
					GVL.A_StepHold := TRUE;
				END_IF;

			// DIGITAL OUTPUT
            E_RobotCmd.CMD_DO_ON:
				// P1 = Output No;
				GVL.Y[step_PRG_A_Interpreter.P1] := TRUE;

                GVL.A_RunStep := GVL.A_RunStep + 1;
                GVL.A_RunState := 0;
				
				// Nếu đang Step Mode thì dừng chờ sau khi chạy xong 1 lệnh
				IF GVL.A_RunMode = 1 THEN
					GVL.A_StepHold := TRUE;
				END_IF;


            E_RobotCmd.CMD_DO_OFF:
                // P1 = Output No;
				GVL.Y[step_PRG_A_Interpreter.P1] := FALSE;

                GVL.A_RunStep := GVL.A_RunStep + 1;
                GVL.A_RunState := 0;
				
				// Nếu đang Step Mode thì dừng chờ sau khi chạy xong 1 lệnh
				IF GVL.A_RunMode = 1 THEN
					GVL.A_StepHold := TRUE;
				END_IF;

			E_RobotCmd.CMD_DO_TOGGLE:
				// P1 = Output No;
				GVL.Y[step_PRG_A_Interpreter.P1] := NOT GVL.Y[step_PRG_A_Interpreter.P1];
				GVL.A_RunStep := GVL.A_RunStep + 1;
				GVL.A_RunState := 0;
				
				// Nếu đang Step Mode thì dừng chờ sau khi chạy xong 1 lệnh
				IF GVL.A_RunMode = 1 THEN
					GVL.A_StepHold := TRUE;
				END_IF;

			 //================================================
			// WAIT
			//================================================
			E_RobotCmd.CMD_WAIT_IN:
				// P1=Input No, P2=Expected 0/1
				IF GVL.X[step_PRG_A_Interpreter.P1] = (step_PRG_A_Interpreter.P2 <> 0) THEN
					GVL.A_RunStep := GVL.A_RunStep + 1;
					GVL.A_RunState := 0;
					// Nếu đang Step Mode thì dừng chờ sau khi chạy xong 1 lệnh
					IF GVL.A_RunMode = 1 THEN
						GVL.A_StepHold := TRUE;
					END_IF;
				END_IF;
			
			E_RobotCmd.CMD_WAIT:
				// P1=Condition No
				IF F_EvalCondition_A(step_PRG_A_Interpreter.P1) THEN
					GVL.A_RunStep := GVL.A_RunStep + 1;
					GVL.A_RunState := 0;
					// Nếu đang Step Mode thì dừng chờ sau khi chạy xong 1 lệnh
					IF GVL.A_RunMode = 1 THEN
						GVL.A_StepHold := TRUE;
					END_IF;
				END_IF;
            
            E_RobotCmd.CMD_Delay:
                // P1 = thời gian delay ms
                tRunDelay(IN := TRUE, PT := INT_TO_TIME(step_PRG_A_Interpreter.P1));

                IF tRunDelay.Q THEN
                    tRunDelay(IN := FALSE);
                    GVL.A_RunStep := GVL.A_RunStep + 1;
                    GVL.A_RunState := 0;
					// Nếu đang Step Mode thì dừng chờ sau khi chạy xong 1 lệnh
					IF GVL.A_RunMode = 1 THEN
						GVL.A_StepHold := TRUE;
					END_IF;
                END_IF;

			//================================================
			// TIMER
			//================================================
			E_RobotCmd.CMD_Timer_Start:
				// P1=Timer No, P2=Time ms
				GVL.A_TimerPT[step_PRG_A_Interpreter.P1] := DINT_TO_TIME(step_PRG_A_Interpreter.P2);
				GVL.A_TimerStart[step_PRG_A_Interpreter.P1] := TRUE;
				GVL.A_TimerDone[step_PRG_A_Interpreter.P1] := FALSE;
	
				GVL.A_RunStep := GVL.A_RunStep + 1;
				GVL.A_RunState := 0;
				
				// Nếu đang Step Mode thì dừng chờ sau khi chạy xong 1 lệnh
				IF GVL.A_RunMode = 1 THEN
					GVL.A_StepHold := TRUE;
				END_IF;
	
	
			E_RobotCmd.CMD_Timer_Wait:
				// P1=Timer No
				IF GVL.A_TimerDone[step_PRG_A_Interpreter.P1] THEN
					GVL.A_TimerStart[step_PRG_A_Interpreter.P1] := FALSE;
					GVL.A_RunStep := GVL.A_RunStep + 1;
					GVL.A_RunState := 0;
					// Nếu đang Step Mode thì dừng chờ sau khi chạy xong 1 lệnh
					IF GVL.A_RunMode = 1 THEN
						GVL.A_StepHold := TRUE;
					END_IF;
				END_IF;
				
			//================================================
			// IF / ELSE
			//================================================
			E_RobotCmd.CMD_IF:
				// P1=Condition No
				IF F_EvalCondition_A(step_PRG_A_Interpreter.P1) THEN
					GVL.A_RunStep := GVL.A_RunStep + 1;
					// Nếu đang Step Mode thì dừng chờ sau khi chạy xong 1 lệnh
					IF GVL.A_RunMode = 1 THEN
						GVL.A_StepHold := TRUE;
					END_IF;
				ELSE
					GVL.A_RunStep := F_FindElseOrEndIf_A(GVL.A_RunStep);
					// Nếu đang Step Mode thì dừng chờ sau khi chạy xong 1 lệnh
					IF GVL.A_RunMode = 1 THEN
						GVL.A_StepHold := TRUE;
					END_IF;
				END_IF;
				GVL.A_RunState := 0;
	
	
			E_RobotCmd.CMD_IF_IN:
				// P1=Input No, P2=Expected 0/1
				IF GVL.X[step_PRG_A_Interpreter.P1] = (step_PRG_A_Interpreter.P2 <> 0) THEN
					GVL.A_RunStep := GVL.A_RunStep + 1;
					// Nếu đang Step Mode thì dừng chờ sau khi chạy xong 1 lệnh
					IF GVL.A_RunMode = 1 THEN
						GVL.A_StepHold := TRUE;
					END_IF;
				ELSE
					GVL.A_RunStep := F_FindElseOrEndIf_A(GVL.A_RunStep);
					// Nếu đang Step Mode thì dừng chờ sau khi chạy xong 1 lệnh
					IF GVL.A_RunMode = 1 THEN
						GVL.A_StepHold := TRUE;
					END_IF;
				END_IF;
				GVL.A_RunState := 0;
	
	
			E_RobotCmd.CMD_IF_VAR:
				// P1=Var No, P2=Operator, P3=SetValue
				IF F_CompareDINT_A(
					Actual := GVL.A_Var[step_PRG_A_Interpreter.P1],
					Operator := step_PRG_A_Interpreter.P2,
					SetValue := step_PRG_A_Interpreter.P3)
				THEN
					GVL.A_RunStep := GVL.A_RunStep + 1;
					// Nếu đang Step Mode thì dừng chờ sau khi chạy xong 1 lệnh
					IF GVL.A_RunMode = 1 THEN
						GVL.A_StepHold := TRUE;
					END_IF;
				ELSE
					GVL.A_RunStep := F_FindElseOrEndIf_A(GVL.A_RunStep);
					// Nếu đang Step Mode thì dừng chờ sau khi chạy xong 1 lệnh
					IF GVL.A_RunMode = 1 THEN
						GVL.A_StepHold := TRUE;
					END_IF;
				END_IF;
				GVL.A_RunState := 0;
	
	
			E_RobotCmd.CMD_IF_REG:
				// P1=Reg No, P2=Operator, P3=SetValue
				IF F_CompareDINT_A(
					Actual := GVL.A_Reg[step_PRG_A_Interpreter.P1],
					Operator := step_PRG_A_Interpreter.P2,
					SetValue := step_PRG_A_Interpreter.P3)
				THEN
					GVL.A_RunStep := GVL.A_RunStep + 1;
					// Nếu đang Step Mode thì dừng chờ sau khi chạy xong 1 lệnh
					IF GVL.A_RunMode = 1 THEN
						GVL.A_StepHold := TRUE;
					END_IF;
				ELSE
					GVL.A_RunStep := F_FindElseOrEndIf_A(GVL.A_RunStep);
					// Nếu đang Step Mode thì dừng chờ sau khi chạy xong 1 lệnh
					IF GVL.A_RunMode = 1 THEN
						GVL.A_StepHold := TRUE;
					END_IF;
				END_IF;
				GVL.A_RunState := 0;
	
	
			E_RobotCmd.CMD_ELSE:
				GVL.A_RunStep := F_FindEndIf_A(GVL.A_RunStep);
				GVL.A_RunState := 0;
				// Nếu đang Step Mode thì dừng chờ sau khi chạy xong 1 lệnh
				IF GVL.A_RunMode = 1 THEN
					GVL.A_StepHold := TRUE;
				END_IF;
	
			E_RobotCmd.CMD_END_IF:
				GVL.A_RunStep := GVL.A_RunStep + 1;
				GVL.A_RunState := 0;
				// Nếu đang Step Mode thì dừng chờ sau khi chạy xong 1 lệnh
				IF GVL.A_RunMode = 1 THEN
					GVL.A_StepHold := TRUE;
				END_IF;
			
			//================================================
			// JUMP / CALL / RETURN
			//================================================
			E_RobotCmd.CMD_JUMP:
				// P1=Target Step
				GVL.A_RunStep := step_PRG_A_Interpreter.P1;
				GVL.A_RunState := 0;
				// Nếu đang Step Mode thì dừng chờ sau khi chạy xong 1 lệnh
				IF GVL.A_RunMode = 1 THEN
					GVL.A_StepHold := TRUE;
				END_IF;
	
	
			E_RobotCmd.CMD_CALL:
				// P1=Target Step
				IF GVL.A_CallStackIndex < 20 THEN
					GVL.A_CallStackIndex := GVL.A_CallStackIndex + 1;
					GVL.A_CallStack[GVL.A_CallStackIndex] := GVL.A_RunStep + 1;
					GVL.A_RunStep := step_PRG_A_Interpreter.P1;
					GVL.A_RunState := 0;
				ELSE
					GVL.A_RunAlarm := TRUE;
					GVL.A_RunAlarmCode := 2101; // Call stack full
					GVL.A_RunErrorStep := GVL.A_RunStep;
					GVL.A_RunState := 900;
				END_IF;
	
	
			E_RobotCmd.CMD_RETURN:
				IF GVL.A_CallStackIndex > 0 THEN
					GVL.A_RunStep := GVL.A_CallStack[GVL.A_CallStackIndex];
					GVL.A_CallStackIndex := GVL.A_CallStackIndex - 1;
					GVL.A_RunState := 0;
				ELSE
					GVL.A_RunAlarm := TRUE;
					GVL.A_RunAlarmCode := 2102; // Return stack empty
					GVL.A_RunErrorStep := GVL.A_RunStep;
					GVL.A_RunState := 900;
				END_IF;
			
			//================================================
			// WHILE
			//================================================
			E_RobotCmd.CMD_WHILE:
				// P1=Condition No
				IF F_EvalCondition_A(step_PRG_A_Interpreter.P1) THEN
					GVL.A_RunStep := GVL.A_RunStep + 1;
					// Nếu đang Step Mode thì dừng chờ sau khi chạy xong 1 lệnh
					IF GVL.A_RunMode = 1 THEN
						GVL.A_StepHold := TRUE;
					END_IF;
				ELSE
					GVL.A_RunStep := F_FindEndWhile_A(GVL.A_RunStep);
					// Nếu đang Step Mode thì dừng chờ sau khi chạy xong 1 lệnh
					IF GVL.A_RunMode = 1 THEN
						GVL.A_StepHold := TRUE;
					END_IF;
				END_IF;
				GVL.A_RunState := 0;
	
	
			E_RobotCmd.CMD_WHILE_IN:
				// P1=Input No, P2=Expected 0/1
				IF GVL.X[step_PRG_A_Interpreter.P1] = (step_PRG_A_Interpreter.P2 <> 0) THEN
					GVL.A_RunStep := GVL.A_RunStep + 1;
					// Nếu đang Step Mode thì dừng chờ sau khi chạy xong 1 lệnh
					IF GVL.A_RunMode = 1 THEN
						GVL.A_StepHold := TRUE;
					END_IF;
				ELSE
					GVL.A_RunStep := F_FindEndWhile_A(GVL.A_RunStep);
					// Nếu đang Step Mode thì dừng chờ sau khi chạy xong 1 lệnh
					IF GVL.A_RunMode = 1 THEN
						GVL.A_StepHold := TRUE;
					END_IF;
				END_IF;
				GVL.A_RunState := 0;
	
	
			E_RobotCmd.CMD_WHILE_REG:
				// P1=Reg No, P2=Operator, P3=SetValue
				IF F_CompareDINT_A(
					Actual := GVL.A_Reg[step_PRG_A_Interpreter.P1],
					Operator := step_PRG_A_Interpreter.P2,
					SetValue := step_PRG_A_Interpreter.P3)
				THEN
					GVL.A_RunStep := GVL.A_RunStep + 1;
					// Nếu đang Step Mode thì dừng chờ sau khi chạy xong 1 lệnh
					IF GVL.A_RunMode = 1 THEN
						GVL.A_StepHold := TRUE;
					END_IF;
				ELSE
					GVL.A_RunStep := F_FindEndWhile_A(GVL.A_RunStep);
					// Nếu đang Step Mode thì dừng chờ sau khi chạy xong 1 lệnh
					IF GVL.A_RunMode = 1 THEN
						GVL.A_StepHold := TRUE;
					END_IF;
				END_IF;
				GVL.A_RunState := 0;
	
	
			E_RobotCmd.CMD_END_WHILE:
// 				GVL.A_RunStep := F_FindWhileStart_A(GVL.A_RunStep);
// 				GVL.A_RunState := 0;

				//--------------------------------------------------------
				// Lưu vị trí WHILE cần quay lại
				//--------------------------------------------------------
				WhileReturnStep :=
					F_FindWhileStart_A(GVL.A_RunStep);

				//--------------------------------------------------------
				// Không nhảy về WHILE ngay.
				// Trước tiên chờ pipeline của vòng hiện tại sạch.
				//--------------------------------------------------------
				GVL.A_RunState := 140;
				
				// Nếu đang Step Mode thì dừng chờ sau khi chạy xong 1 lệnh
				IF GVL.A_RunMode = 1 THEN
					GVL.A_StepHold := TRUE;
				END_IF;
			
// 			//================================================
// 			// VISION
// 			//================================================
// 			E_RobotCmd.CMD_VISION_TRIGGER:
// 				GVL.A_VisionTriggerReq := TRUE;
// 				GVL.A_RunStep := GVL.A_RunStep + 1;
// 				GVL.A_RunState := 0;
// 				// Nếu đang Step Mode thì dừng chờ sau khi chạy xong 1 lệnh
// 				IF GVL.A_RunMode = 1 THEN
// 					GVL.A_StepHold := TRUE;
// 				END_IF;

			E_RobotCmd.CMD_VISION_TRIGGER:
				//=========================================================================
				// VISION TRIGGER - ROBOT A
				//-------------------------------------------------------------------------
				// Command này thực hiện toàn bộ transaction:
				//
				// Robot A -> Vision Manager -> FB_VisionAlign -> Vision
				//
				// P1 = CameraID.
				// P2 = JobID.
				// P3 = A_Var index nhận business result.
				//
				// A_Var[P3] = 1 : Vision Result OK.
				// A_Var[P3] = 0 : Vision Result NG / NOT_FOUND / LOW_SCORE / ...
				//
				// Lỗi communication/config/protocol/timeout:
				// -> A_VisionError = TRUE.
				// -> Robot Alarm.
				// -> Không chuyển sang step tiếp theo.
				//=========================================================================
			
			
				//=========================================================================
				// 1. START COMMAND
				// Chỉ thực hiện một lần khi command Vision chưa active.
				//=========================================================================
				IF NOT xVisionStepActiveA THEN
			
					//---------------------------------------------------------------------
					// Latch tham số command.
					//---------------------------------------------------------------------
					uiVisionCameraIDA := INT_TO_UINT(step_PRG_A_Interpreter.P1);
					uiVisionJobIDA := INT_TO_UINT(step_PRG_A_Interpreter.P2);
					iVisionResultVarA := DINT_TO_INT(step_PRG_A_Interpreter.P3);
			
					//---------------------------------------------------------------------
					// Kiểm tra CameraID trước khi gửi Request.
					//---------------------------------------------------------------------
					IF (uiVisionCameraIDA < 1)
					OR (uiVisionCameraIDA > GVL.C_MAX_VISION_CHANNELS) THEN
			
						GVL.A_VisionDone := FALSE;
						GVL.A_VisionOK := FALSE;
						GVL.A_VisionError := TRUE;
			
						GVL.A_RunAlarm := TRUE;
						GVL.A_RunAlarmCode := 2201;
						GVL.A_RunErrorStep := GVL.A_RunStep;
						GVL.A_RunState := 900;
			
					//---------------------------------------------------------------------
					// A_Var của project hiện tại có index 0..200.
					//---------------------------------------------------------------------
					ELSIF (iVisionResultVarA < 0)
					OR (iVisionResultVarA > 200) THEN
			
						GVL.A_VisionDone := FALSE;
						GVL.A_VisionOK := FALSE;
						GVL.A_VisionError := TRUE;
			
						GVL.A_RunAlarm := TRUE;
						GVL.A_RunAlarmCode := 2202;
						GVL.A_RunErrorStep := GVL.A_RunStep;
						GVL.A_RunState := 900;
			
					ELSE
						//-----------------------------------------------------------------
						// Xóa business result cũ.
						//-----------------------------------------------------------------
						GVL.A_Var[iVisionResultVarA] := 0;
			
						//-----------------------------------------------------------------
						// Xóa status tương thích logic Robot cũ.
						//-----------------------------------------------------------------
						GVL.A_VisionDone := FALSE;
						GVL.A_VisionOK := FALSE;
						GVL.A_VisionError := FALSE;
			
						//-----------------------------------------------------------------
						// Gửi Request sang Vision Manager.
						//
						// CameraID và JobID phải được ghi TRƯỚC Execute.
						//-----------------------------------------------------------------
						GVL.g_stVisionAlignRequestA.CameraID := uiVisionCameraIDA;
						GVL.g_stVisionAlignRequestA.JobID := uiVisionJobIDA;
						GVL.g_stVisionAlignRequestA.Execute := TRUE;
			
						//-----------------------------------------------------------------
						// Đánh dấu command Vision của Robot A đang hoạt động.
						//-----------------------------------------------------------------
						xVisionStepActiveA := TRUE;
					END_IF;
				END_IF;
			
			
				//=========================================================================
				// 2. WAIT TRANSACTION DONE
				//=========================================================================
				IF xVisionStepActiveA AND GVL.g_stVisionAlignRequestA.Done THEN
			
					//---------------------------------------------------------------------
					// Vision transaction hoàn thành bình thường.
					//
					// ResultOK quyết định business result:
					// TRUE  -> A_Var[P3] = 1.
					// FALSE -> A_Var[P3] = 0.
					//---------------------------------------------------------------------
					IF GVL.g_stVisionAlignRequestA.ResultOK THEN
						GVL.A_Var[iVisionResultVarA] := 1;
						GVL.A_VisionOK := TRUE;
					ELSE
						GVL.A_Var[iVisionResultVarA] := 0;
						GVL.A_VisionOK := FALSE;
					END_IF;
			
					//---------------------------------------------------------------------
					// Transaction đã hoàn thành.
					//---------------------------------------------------------------------
					GVL.A_VisionDone := TRUE;
					GVL.A_VisionError := FALSE;
			
					//---------------------------------------------------------------------
					// Hạ Execute = ACK từ Robot về Manager.
					//
					// Manager thấy Execute FALSE sẽ:
					// - Reset Done.
					// - Giải phóng Camera.
					// - Đưa Camera về State 0.
					//---------------------------------------------------------------------
					GVL.g_stVisionAlignRequestA.Execute := FALSE;
			
					//---------------------------------------------------------------------
					// Kết thúc command local.
					//---------------------------------------------------------------------
					xVisionStepActiveA := FALSE;
			
					//---------------------------------------------------------------------
					// Chuyển sang command tiếp theo.
					//---------------------------------------------------------------------
					GVL.A_RunStep := GVL.A_RunStep + 1;
					GVL.A_RunState := 0;
			
					//---------------------------------------------------------------------
					// Step Mode: giữ chương trình sau khi hoàn thành một command.
					//---------------------------------------------------------------------
					IF GVL.A_RunMode = 1 THEN
						GVL.A_StepHold := TRUE;
					END_IF;
			
			
				//=========================================================================
				// 3. WAIT TRANSACTION ERROR
				//=========================================================================
				ELSIF xVisionStepActiveA AND GVL.g_stVisionAlignRequestA.Error THEN
				
					// LƯU MÃ LỖI TRƯỚC KHI HẠ EXECUTE.
					// Manager sẽ reset ErrorID sau khi Execute = FALSE.
					iVisionErrorIDA := GVL.g_stVisionAlignRequestA.ErrorID;
				
					// Không sử dụng kết quả Vision khi transaction lỗi.
					GVL.A_Var[iVisionResultVarA] := 0;
					GVL.A_VisionDone := FALSE;
					GVL.A_VisionOK := FALSE;
					GVL.A_VisionError := TRUE;
				
					// Báo Alarm Robot.
					GVL.A_RunAlarm := TRUE;
					GVL.A_RunAlarmCode := 2201;
					GVL.A_RunErrorStep := GVL.A_RunStep;
					GVL.A_RunState := 900;
				
					// Kết thúc command Vision local.
					xVisionStepActiveA := FALSE;
				
					// Hạ Execute CUỐI CÙNG.
					// Manager nhận ACK này và sau đó mới reset Request.
					GVL.g_stVisionAlignRequestA.Execute := FALSE;
				
				END_IF;
							
	
			E_RobotCmd.CMD_VISION_SET_POINT:

				//=========================================================================
				// VISION SET POINT
				//-------------------------------------------------------------------------
				// P1 = Master Point No.
				// P2 = Destination Point No.
				// P3 = Vision Result Index.
				//
				// Destination = Master + Vision Result[P3]
				//
				// Ví dụ:
				// VISION_SET_POINT P10 P101 1
				// VISION_SET_POINT P10 P102 2
				//
				// P101 = P10 + Result[1]
				// P102 = P10 + Result[2]
				//
				// Chỉ yêu cầu Header của Vision Result hợp lệ.
				// Không kiểm tra ObjectCount.
				// Không kiểm tra Object.Valid.
				// Không kiểm tra Vision có trả đủ số lượng Object hay không.
				//=========================================================================
			
				//-------------------------------------------------------------------------
				// 1. KIỂM TRA MASTER / DESTINATION POINT
				//-------------------------------------------------------------------------
				IF (step_PRG_A_Interpreter.P1 < 1) OR (step_PRG_A_Interpreter.P1 > 500)
				OR (step_PRG_A_Interpreter.P2 < 1) OR (step_PRG_A_Interpreter.P2 > 500)
				OR (step_PRG_A_Interpreter.P1 = step_PRG_A_Interpreter.P2) THEN
			
					GVL.A_RunAlarm := TRUE;
					GVL.A_RunAlarmCode := 2203;      // Master/Destination Point không hợp lệ.
					GVL.A_RunErrorStep := GVL.A_RunStep;
					GVL.A_RunState := 900;
			
				//-------------------------------------------------------------------------
				// 2. KIỂM TRA RESULT INDEX
				//-------------------------------------------------------------------------
				ELSIF (step_PRG_A_Interpreter.P3 < 1)
				OR (step_PRG_A_Interpreter.P3 > GVL.C_MAX_VISION_TRACK_OBJECTS_PER_FRAME) THEN
			
					GVL.A_RunAlarm := TRUE;
					GVL.A_RunAlarmCode := 2205;      // Vision Result Index ngoài vùng Array.
					GVL.A_RunErrorStep := GVL.A_RunStep;
					GVL.A_RunState := 900;
			
				//-------------------------------------------------------------------------
				// 3. CHỈ KIỂM TRA HEADER
				//-------------------------------------------------------------------------
				ELSIF NOT GVL.g_aVisionResult[uiVisionCameraIDA].Header.Valid THEN
			
					GVL.A_RunAlarm := TRUE;
					GVL.A_RunAlarmCode := 2204;      // Vision Header không hợp lệ.
					GVL.A_RunErrorStep := GVL.A_RunStep;
					GVL.A_RunState := 900;
			
				ELSE
			
					//=====================================================================
					// 4. DESTINATION = MASTER + VISION RESULT[P3]
					//=====================================================================
			
					// X
					GVL_1.DATA_RB_A.X_POS[DINT_TO_INT(step_PRG_A_Interpreter.P2)] :=
						GVL_1.DATA_RB_A.X_POS[DINT_TO_INT(step_PRG_A_Interpreter.P1)]
						+ GVL.g_aVisionResult[uiVisionCameraIDA].TrackObjectResult.Objects[DINT_TO_UINT(step_PRG_A_Interpreter.P3)].Pos.X;
			
					// Y
					GVL_1.DATA_RB_A.Y_POS[DINT_TO_INT(step_PRG_A_Interpreter.P2)] :=
						GVL_1.DATA_RB_A.Y_POS[DINT_TO_INT(step_PRG_A_Interpreter.P1)]
						+ GVL.g_aVisionResult[uiVisionCameraIDA].TrackObjectResult.Objects[DINT_TO_UINT(step_PRG_A_Interpreter.P3)].Pos.Y;
			
					// Z
					GVL_1.DATA_RB_A.Z_POS[DINT_TO_INT(step_PRG_A_Interpreter.P2)] :=
						GVL_1.DATA_RB_A.Z_POS[DINT_TO_INT(step_PRG_A_Interpreter.P1)]
						+ GVL.g_aVisionResult[uiVisionCameraIDA].TrackObjectResult.Objects[DINT_TO_UINT(step_PRG_A_Interpreter.P3)].Pos.Z;
			
					// R
					GVL_1.DATA_RB_A.R_POS[DINT_TO_INT(step_PRG_A_Interpreter.P2)] :=
						GVL_1.DATA_RB_A.R_POS[DINT_TO_INT(step_PRG_A_Interpreter.P1)]
						+ GVL.g_aVisionResult[uiVisionCameraIDA].TrackObjectResult.Objects[DINT_TO_UINT(step_PRG_A_Interpreter.P3)].Pos.A;
			
					//=====================================================================
					// 5. COMMAND HOÀN THÀNH
					//=====================================================================
					GVL.A_RunStep := GVL.A_RunStep + 1;
					GVL.A_RunState := 0;
			
					IF GVL.A_RunMode = 1 THEN
						GVL.A_StepHold := TRUE;
					END_IF;
			
				END_IF;
	
	
			E_RobotCmd.CMD_VISION_PICK:

				//=========================================================================
				// VISION PICK
				//-------------------------------------------------------------------------
				// Hiện tại mới xác nhận Result Vision tồn tại.
				// Phần Camera->Robot Transform và tạo Target Pick sẽ bổ sung sau.
				//=========================================================================
			
				IF GVL.A_VisionHeaderOK THEN
					GVL.A_RunStep := GVL.A_RunStep + 1;
					GVL.A_RunState := 0;
			
					IF GVL.A_RunMode = 1 THEN
						GVL.A_StepHold := TRUE;
					END_IF;
			
				ELSE
					GVL.A_RunAlarm := TRUE;
					GVL.A_RunAlarmCode := 2202;
					GVL.A_RunErrorStep := GVL.A_RunStep;
					GVL.A_RunState := 900;
				END_IF;
	
	
			E_RobotCmd.CMD_VISION_CHECK:

				//=========================================================================
				// CHECK LAST VISION RESULT
				//-------------------------------------------------------------------------
				// TRUE  -> chạy Step tiếp theo.
				// FALSE -> nhảy tới ELSE / END_IF.
				//=========================================================================
			
				IF GVL.A_VisionHeaderOK THEN
					GVL.A_RunStep := GVL.A_RunStep + 1;
				ELSE
					GVL.A_RunStep := F_FindElseOrEndIf_A(GVL.A_RunStep);
				END_IF;
			
				GVL.A_RunState := 0;
			
				IF GVL.A_RunMode = 1 THEN
					GVL.A_StepHold := TRUE;
				END_IF;
			
			//================================================
			// TRACKING
			//================================================
			E_RobotCmd.CMD_TRACK_ON:
				GVL.A_TrackEnable := TRUE;
				GVL.A_RunStep := GVL.A_RunStep + 1;
				GVL.A_RunState := 0;
	
	
			E_RobotCmd.CMD_TRACK_OFF:
				GVL.A_TrackEnable := FALSE;
				GVL.A_RunStep := GVL.A_RunStep + 1;
				GVL.A_RunState := 0;
	
	
			//==========================================================================
			// TRACK PICK
			//--------------------------------------------------------------------------
			// P1 = RecipeID
			// P2 = Target Pick Count
			// P3 = Tool Mask
			//
			// Ví dụ:
			// P1=1, P2=1, P3=1 -> Recipe 1, Pick 1, chỉ Tool 1.
			// P1=1, P2=2, P3=3 -> Recipe 1, Pick 2, Tool 1 + Tool 2.
			//==========================================================================
			E_RobotCmd.CMD_TRACK_PICK:
			
				//----------------------------------------------------------------------
				// 1. CHỈ PHÁT COMMAND MỘT LẦN
				//----------------------------------------------------------------------
				IF NOT GVL.A_StepActive THEN
			
					// Chỉ bắt đầu khi Motion Pipeline trước đó đã sạch.
					IF (GVL.A_MotionCount <= 0)
					AND (GVL.A_ActiveMotionCount <= 0)
					AND NOT GVL.A_MotionManagerBusy THEN
			
						//--------------------------------------------------------------
						// Tạo CommandID mới.
						//--------------------------------------------------------------
						GVL.g_stMultiTrackCommandA.CommandID :=
							GVL.g_stMultiTrackCommandA.CommandID + 1;
			
						IF GVL.g_stMultiTrackCommandA.CommandID = 0 THEN
							GVL.g_stMultiTrackCommandA.CommandID := 1;
						END_IF;
			
						//--------------------------------------------------------------
						// Nạp tham số từ dòng Interpreter.
						//--------------------------------------------------------------
						GVL.g_stMultiTrackCommandA.RecipeID :=
							INT_TO_UINT(step_PRG_A_Interpreter.P1);
			
						GVL.g_stMultiTrackCommandA.TargetPickCountOverride :=
							INT_TO_UINT(step_PRG_A_Interpreter.P2);
			
						GVL.g_stMultiTrackCommandA.ToolMaskOverride :=
							DINT_TO_DWORD(step_PRG_A_Interpreter.P3);
			
						//--------------------------------------------------------------
						// Command mới.
						//--------------------------------------------------------------
						GVL.g_stMultiTrackCommandA.Reset := FALSE;
						GVL.g_stMultiTrackCommandA.Abort := FALSE;
						GVL.g_stMultiTrackCommandA.Execute := TRUE;
			
						//--------------------------------------------------------------
						// Nhớ CommandID mà Interpreter đang chờ.
						//--------------------------------------------------------------
						udiTrackCommandIDA :=
							GVL.g_stMultiTrackCommandA.CommandID;
			
						//--------------------------------------------------------------
						// Không phát lại command ở scan tiếp theo.
						//--------------------------------------------------------------
						GVL.A_StepActive := TRUE;
			
					END_IF;
			
				END_IF;
			
			
				//----------------------------------------------------------------------
				// 2. TRACKING HOÀN THÀNH ĐÚNG COMMAND
				//----------------------------------------------------------------------
				IF GVL.A_StepActive
				AND GVL.g_xTrackOKA
				AND GVL.g_udiTrackDoneCommandIDA = udiTrackCommandIDA THEN
			
					// Hạ Execute sau khi Application hoàn thành.
					GVL.g_stMultiTrackCommandA.Execute := FALSE;
			
					// Kết thúc transaction của Interpreter.
					GVL.A_StepActive := FALSE;
					udiTrackCommandIDA := 0;
			
					// Sang dòng chương trình tiếp theo.
					GVL.A_RunStep := GVL.A_RunStep + 1;
					GVL.A_RunState := 0;
			
					// Step Mode: dừng sau khi hoàn thành TRACK_PICK.
					IF GVL.A_RunMode = 1 THEN
						GVL.A_StepHold := TRUE;
					END_IF;
			
				//----------------------------------------------------------------------
				// 3. TRACKING ERROR
				//----------------------------------------------------------------------
				ELSIF GVL.A_StepActive
				AND GVL.g_xTrackErrorA THEN
			
					GVL.g_stMultiTrackCommandA.Execute := FALSE;
			
					GVL.A_StepActive := FALSE;
					udiTrackCommandIDA := 0;
			
					GVL.A_RunAlarm := TRUE;
					GVL.A_RunAlarmCode :=
						UDINT_TO_INT(GVL.g_udiTrackErrorIDA);
			
					GVL.A_RunErrorStep := GVL.A_RunStep;
					GVL.A_RunState := 900;
			
				END_IF;
			
			//=========================================================================
			// TOOL RELEASE
			//-------------------------------------------------------------------------
			// P1 = ToolID cần nhả sản phẩm.
			//=========================================================================
			E_RobotCmd.CMD_TOOL_RELEASE:
			
				//---------------------------------------------------------------------
				// 1. PHÁT LỆNH RELEASE MỘT LẦN
				//---------------------------------------------------------------------
				IF NOT GVL.A_StepActive THEN
			
					// Kiểm tra ToolID hợp lệ.
					IF (step_PRG_A_Interpreter.P1 >= 1)
					AND (step_PRG_A_Interpreter.P1 <= GVL.C_MAX_TOOLS) THEN
			
						//-------------------------------------------------------------
						// Chỉ Release Tool đang thực sự giữ sản phẩm.
						//-------------------------------------------------------------
						IF GVL.g_aToolStatusA[step_PRG_A_Interpreter.P1].Occupied THEN
			
							//---------------------------------------------------------
							// Tạo CommandID mới.
							//---------------------------------------------------------
							GVL.g_stInterpreterToolCommandA.CommandID :=
								GVL.g_stInterpreterToolCommandA.CommandID + 1;
			
							IF GVL.g_stInterpreterToolCommandA.CommandID = 0 THEN
								GVL.g_stInterpreterToolCommandA.CommandID := 1;
							END_IF;
			
							//---------------------------------------------------------
							// Nạp command.
							//---------------------------------------------------------
							GVL.g_stInterpreterToolCommandA.ToolID :=
								INT_TO_UINT(step_PRG_A_Interpreter.P1);
			
							GVL.g_stInterpreterToolCommandA.CommandType :=
								E_ToolCommandType.RELEASE;
			
							// Giữ ObjectID hiện tại để debug/trace.
							GVL.g_stInterpreterToolCommandA.ObjectID :=
								GVL.g_aToolStatusA[step_PRG_A_Interpreter.P1].HeldObjectID;
			
							GVL.g_stInterpreterToolCommandA.Reset := FALSE;
							GVL.g_stInterpreterToolCommandA.Abort := FALSE;
							GVL.g_stInterpreterToolCommandA.Execute := TRUE;
			
							//---------------------------------------------------------
							// Nhớ CommandID đang chờ.
							//---------------------------------------------------------
							udiToolReleaseCommandIDA :=
								GVL.g_stInterpreterToolCommandA.CommandID;
			
							GVL.A_StepActive := TRUE;
			
						ELSE
			
							//---------------------------------------------------------
							// Tool không giữ vật -> coi là lỗi dạy chương trình.
							//---------------------------------------------------------
							GVL.A_RunAlarm := TRUE;
							GVL.A_RunAlarmCode := 2502;
							GVL.A_RunErrorStep := GVL.A_RunStep;
							GVL.A_RunState := 900;
			
						END_IF;
			
					ELSE
			
						//-------------------------------------------------------------
						// ToolID ngoài phạm vi.
						//-------------------------------------------------------------
						GVL.A_RunAlarm := TRUE;
						GVL.A_RunAlarmCode := 2501;
						GVL.A_RunErrorStep := GVL.A_RunStep;
						GVL.A_RunState := 900;
			
					END_IF;
			
				END_IF;
			
			
				//---------------------------------------------------------------------
				// 2. RELEASE HOÀN THÀNH
				//---------------------------------------------------------------------
				IF GVL.A_StepActive
				AND GVL.g_aToolStatusA[step_PRG_A_Interpreter.P1].Done
				AND GVL.g_aToolStatusA[step_PRG_A_Interpreter.P1].ResponseCommandID
					= udiToolReleaseCommandIDA THEN
			
					//-------------------------------------------------------------
					// Hạ Execute để tạo lại cạnh cho command sau.
					//-------------------------------------------------------------
					GVL.g_stInterpreterToolCommandA.Execute := FALSE;
			
					GVL.A_StepActive := FALSE;
					udiToolReleaseCommandIDA := 0;
			
					//-------------------------------------------------------------
					// Sang step kế tiếp.
					//-------------------------------------------------------------
					GVL.A_RunStep := GVL.A_RunStep + 1;
					GVL.A_RunState := 0;
			
					IF GVL.A_RunMode = 1 THEN
						GVL.A_StepHold := TRUE;
					END_IF;
			
			
				//---------------------------------------------------------------------
				// 3. TOOL ERROR
				//---------------------------------------------------------------------
				ELSIF GVL.A_StepActive
				AND GVL.g_aToolStatusA[step_PRG_A_Interpreter.P1].Error THEN
			
					GVL.g_stInterpreterToolCommandA.Execute := FALSE;
			
					GVL.A_StepActive := FALSE;
					udiToolReleaseCommandIDA := 0;
			
					GVL.A_RunAlarm := TRUE;
			
					GVL.A_RunAlarmCode :=
						UDINT_TO_INT(
							GVL.g_aToolStatusA[step_PRG_A_Interpreter.P1].ErrorID
						);
			
					GVL.A_RunErrorStep := GVL.A_RunStep;
					GVL.A_RunState := 900;
			
				END_IF;
	

			E_RobotCmd.CMD_TRACK_PLACE:
				GVL.A_TrackPlaceReq := TRUE;
	
				IF GVL.A_TrackPlaceDone THEN
					GVL.A_TrackPlaceReq := FALSE;
					GVL.A_RunStep := GVL.A_RunStep + 1;
					GVL.A_RunState := 0;
				END_IF;
				
			E_RobotCmd.CMD_CONV_PICK:

// 				// Không bắt đầu Application khi pipeline motion cũ còn hoạt động.
// 				IF NOT GVL.A_StepActive THEN
// 					IF GVL.A_MotionCount = 0 AND GVL.A_ActiveMotionCount = 0 THEN
// 						GVL.g_stApplicationCommandA.ApplicationID := E_ApplicationID.APP_CONVEYOR_PICK;
// 						GVL.g_stApplicationCommandA.RecipeID := TO_UINT(step.P1);
// 						GVL.g_stApplicationCommandA.RobotID := 1;
// 						GVL.g_stApplicationCommandA.CommandID := GVL.g_stApplicationCommandA.CommandID + 1;
// 						GVL.g_stApplicationCommandA.Execute := TRUE;
// 						GVL.A_StepActive := TRUE;
// 					END_IF;
// 				END_IF;
// 			
// 				// Application hoàn thành: hạ Execute và chuyển step.
// 				IF GVL.g_stApplicationResponseA.Done THEN
// 					GVL.g_stApplicationCommandA.Execute := FALSE;
// 					GVL.A_StepActive := FALSE;
// 					GVL.A_RunStep := GVL.A_RunStep + 1;
// 				END_IF;
// 			
// 				// Application lỗi: dừng Interpreter.
// 				IF GVL.g_stApplicationResponseA.Error THEN
// 					GVL.g_stApplicationCommandA.Execute := FALSE;
// 					GVL.A_StepActive := FALSE;
// 					GVL.A_RunAlarm := TRUE;
// 					GVL.A_RunAlarmCode := TO_INT(GVL.g_stApplicationResponseA.ErrorID);
// 					GVL.A_RunErrorStep := GVL.A_RunStep;
// 				END_IF;

				// Chỉ bắt đầu khi Motion Queue và các slot hiện tại đã sạch.
				IF NOT GVL.A_StepActive THEN
					IF GVL.A_MotionCount = 0 AND GVL.A_ActiveMotionCount = 0 THEN
						GVL.A_TrackStartCmd := TRUE;
						GVL.A_StepActive := TRUE;
					END_IF;
				END_IF;
			
				// Sau khi engine nhận cạnh Start, hạ request.
				IF GVL.A_TrackEngineBusy THEN
					GVL.A_TrackStartCmd := FALSE;
				END_IF;
			
				// Hoàn thành application thì tăng step.
				IF GVL.A_TrackEngineDone THEN
					GVL.A_TrackStartCmd := FALSE;
					GVL.A_StepActive := FALSE;
					GVL.A_RunStep := GVL.A_RunStep + 1;
					GVL.A_RunState := 0;
				END_IF;
			
				// Lỗi application thì dừng Interpreter.
				IF GVL.A_TrackEngineError THEN
					GVL.A_TrackStartCmd := FALSE;
					GVL.A_StepActive := FALSE;
					GVL.A_RunAlarm := TRUE;
					GVL.A_RunAlarmCode := TO_INT(GVL.A_TrackEngineErrorID);
					GVL.A_RunErrorStep := GVL.A_RunStep;
				END_IF;

			//=========================================================================
			// MODBUS / POINT COMMANDS - ROBOT A
			//=========================================================================
			
			E_RobotCmd.CMD_MB_REG_READ:
				// P1 = MODBUS Index [0..1999]
				// P2 = A_Reg Destination [1..200]
				// GVL.MODBUS[] dùng chung
				// Giá trị MODBUS được hiểu là INT16 có dấu
			
				IF (step_PRG_A_Interpreter.P1 >= 0) AND (step_PRG_A_Interpreter.P1 <= 1999)
				AND (step_PRG_A_Interpreter.P2 >= 1) AND (step_PRG_A_Interpreter.P2 <= 200) THEN
			
					GVL.A_Reg[step_PRG_A_Interpreter.P2] := INT_TO_DINT(WORD_TO_INT(GVL.MODBUS[step_PRG_A_Interpreter.P1]));
			
					GVL.A_RunStep := GVL.A_RunStep + 1;
					GVL.A_RunState := 0;
					IF GVL.A_RunMode = 1 THEN GVL.A_StepHold := TRUE; END_IF;
			
				ELSE
					GVL.A_RunAlarm := TRUE;
					GVL.A_RunAlarmCode := 2503;
					GVL.A_RunErrorStep := GVL.A_RunStep;
					GVL.A_RunState := 900;
				END_IF;
			
			//-------------------------------------------------------------------------
			// CMD_MB_REG_SET
			// P1 = MODBUS Index [0..1999]
			// P2 = Giá trị INT16 signed [-32768..32767]
			//-------------------------------------------------------------------------
			E_RobotCmd.CMD_MB_REG_SET:
				IF (step_PRG_A_Interpreter.P1 >= 0) AND (step_PRG_A_Interpreter.P1 <= 1999) THEN
					GVL.MODBUS[step_PRG_A_Interpreter.P1] := INT_TO_WORD(step_PRG_A_Interpreter.P2);
			
					GVL.A_RunStep := GVL.A_RunStep + 1;
					GVL.A_RunState := 0;
					IF GVL.A_RunMode = 1 THEN GVL.A_StepHold := TRUE; END_IF;
				ELSE
					GVL.A_RunAlarm := TRUE;
					GVL.A_RunAlarmCode := 2501; // MODBUS index invalid
					GVL.A_RunErrorStep := GVL.A_RunStep;
					GVL.A_RunState := 900;
				END_IF;
			
			
			//-------------------------------------------------------------------------
			// CMD_MB_BIT_SET
			// P1 = MODBUS Index [0..1999]
			// P2 = Bit Index [0..15]
			// P3 = 0: Reset bit / <>0: Set bit
			//-------------------------------------------------------------------------
			E_RobotCmd.CMD_MB_BIT_SET:
				IF (step_PRG_A_Interpreter.P1 >= 0) AND (step_PRG_A_Interpreter.P1 <= 1999)
				AND (step_PRG_A_Interpreter.P2 >= 0) AND (step_PRG_A_Interpreter.P2 <= 15) THEN
			
					IF step_PRG_A_Interpreter.P3 <> 0 THEN
						GVL.MODBUS[step_PRG_A_Interpreter.P1] := GVL.MODBUS[step_PRG_A_Interpreter.P1] OR SHL(WORD#1, step_PRG_A_Interpreter.P2);
					ELSE
						GVL.MODBUS[step_PRG_A_Interpreter.P1] := GVL.MODBUS[step_PRG_A_Interpreter.P1] AND NOT SHL(WORD#1, step_PRG_A_Interpreter.P2);
					END_IF;
			
					GVL.A_RunStep := GVL.A_RunStep + 1;
					GVL.A_RunState := 0;
					IF GVL.A_RunMode = 1 THEN GVL.A_StepHold := TRUE; END_IF;
				ELSE
					GVL.A_RunAlarm := TRUE;
					GVL.A_RunAlarmCode := 2502; // MODBUS index/bit invalid
					GVL.A_RunErrorStep := GVL.A_RunStep;
					GVL.A_RunState := 900;
				END_IF;
			
			
			//=========================================================================
			// POINT CALCULATION COMMANDS - ROBOT A
			//=========================================================================
			
			//-------------------------------------------------------------------------
			// POINT COPY
			// P1 = Destination Point
			// P2 = Source Point
			// Dest := Source
			//-------------------------------------------------------------------------
			E_RobotCmd.CMD_POINT_COPY:
				IF (step_PRG_A_Interpreter.P1 >= 1) AND (step_PRG_A_Interpreter.P1 <= 500)
				AND (step_PRG_A_Interpreter.P2 >= 1) AND (step_PRG_A_Interpreter.P2 <= 500) THEN
			
					GVL_1.DATA_RB_A.X_POS[step_PRG_A_Interpreter.P1] := GVL_1.DATA_RB_A.X_POS[step_PRG_A_Interpreter.P2];
					GVL_1.DATA_RB_A.Y_POS[step_PRG_A_Interpreter.P1] := GVL_1.DATA_RB_A.Y_POS[step_PRG_A_Interpreter.P2];
					GVL_1.DATA_RB_A.Z_POS[step_PRG_A_Interpreter.P1] := GVL_1.DATA_RB_A.Z_POS[step_PRG_A_Interpreter.P2];
					GVL_1.DATA_RB_A.R_POS[step_PRG_A_Interpreter.P1] := GVL_1.DATA_RB_A.R_POS[step_PRG_A_Interpreter.P2];
			
					GVL.A_RunStep := GVL.A_RunStep + 1;
					GVL.A_RunState := 0;
					IF GVL.A_RunMode = 1 THEN
						GVL.A_StepHold := TRUE;
					END_IF;
			
				ELSE
					GVL.A_RunAlarm := TRUE;
					GVL.A_RunAlarmCode := 2510; // Point index invalid
					GVL.A_RunErrorStep := GVL.A_RunStep;
					GVL.A_RunState := 900;
				END_IF;
			
			
			//-------------------------------------------------------------------------
			// POINT ADD
			// P1 = Destination Point
			// P2 = Base Point
			// P3 = Offset Point
			// Dest := Base + Offset
			//-------------------------------------------------------------------------
			E_RobotCmd.CMD_POINT_ADD:
				IF (step_PRG_A_Interpreter.P1 >= 1) AND (step_PRG_A_Interpreter.P1 <= 500)
				AND (step_PRG_A_Interpreter.P2 >= 1) AND (step_PRG_A_Interpreter.P2 <= 500)
				AND (step_PRG_A_Interpreter.P3 >= 1) AND (step_PRG_A_Interpreter.P3 <= 500) THEN
			
					GVL_1.DATA_RB_A.X_POS[step_PRG_A_Interpreter.P1] := GVL_1.DATA_RB_A.X_POS[step_PRG_A_Interpreter.P2] + GVL_1.DATA_RB_A.X_POS[step_PRG_A_Interpreter.P3];
					GVL_1.DATA_RB_A.Y_POS[step_PRG_A_Interpreter.P1] := GVL_1.DATA_RB_A.Y_POS[step_PRG_A_Interpreter.P2] + GVL_1.DATA_RB_A.Y_POS[step_PRG_A_Interpreter.P3];
					GVL_1.DATA_RB_A.Z_POS[step_PRG_A_Interpreter.P1] := GVL_1.DATA_RB_A.Z_POS[step_PRG_A_Interpreter.P2] + GVL_1.DATA_RB_A.Z_POS[step_PRG_A_Interpreter.P3];
					GVL_1.DATA_RB_A.R_POS[step_PRG_A_Interpreter.P1] := GVL_1.DATA_RB_A.R_POS[step_PRG_A_Interpreter.P2] + GVL_1.DATA_RB_A.R_POS[step_PRG_A_Interpreter.P3];
			
					GVL.A_RunStep := GVL.A_RunStep + 1;
					GVL.A_RunState := 0;
					IF GVL.A_RunMode = 1 THEN
						GVL.A_StepHold := TRUE;
					END_IF;
			
				ELSE
					GVL.A_RunAlarm := TRUE;
					GVL.A_RunAlarmCode := 2511; // Point index invalid
					GVL.A_RunErrorStep := GVL.A_RunStep;
					GVL.A_RunState := 900;
				END_IF;
			
			
			//-------------------------------------------------------------------------
			// POINT SUB
			// P1 = Destination Point
			// P2 = Base Point
			// P3 = Offset Point
			// Dest := Base - Offset
			//-------------------------------------------------------------------------
			E_RobotCmd.CMD_POINT_SUB:
				IF (step_PRG_A_Interpreter.P1 >= 1) AND (step_PRG_A_Interpreter.P1 <= 500)
				AND (step_PRG_A_Interpreter.P2 >= 1) AND (step_PRG_A_Interpreter.P2 <= 500)
				AND (step_PRG_A_Interpreter.P3 >= 1) AND (step_PRG_A_Interpreter.P3 <= 500) THEN
			
					GVL_1.DATA_RB_A.X_POS[step_PRG_A_Interpreter.P1] := GVL_1.DATA_RB_A.X_POS[step_PRG_A_Interpreter.P2] - GVL_1.DATA_RB_A.X_POS[step_PRG_A_Interpreter.P3];
					GVL_1.DATA_RB_A.Y_POS[step_PRG_A_Interpreter.P1] := GVL_1.DATA_RB_A.Y_POS[step_PRG_A_Interpreter.P2] - GVL_1.DATA_RB_A.Y_POS[step_PRG_A_Interpreter.P3];
					GVL_1.DATA_RB_A.Z_POS[step_PRG_A_Interpreter.P1] := GVL_1.DATA_RB_A.Z_POS[step_PRG_A_Interpreter.P2] - GVL_1.DATA_RB_A.Z_POS[step_PRG_A_Interpreter.P3];
					GVL_1.DATA_RB_A.R_POS[step_PRG_A_Interpreter.P1] := GVL_1.DATA_RB_A.R_POS[step_PRG_A_Interpreter.P2] - GVL_1.DATA_RB_A.R_POS[step_PRG_A_Interpreter.P3];
			
					GVL.A_RunStep := GVL.A_RunStep + 1;
					GVL.A_RunState := 0;
					IF GVL.A_RunMode = 1 THEN
						GVL.A_StepHold := TRUE;
					END_IF;
			
				ELSE
					GVL.A_RunAlarm := TRUE;
					GVL.A_RunAlarmCode := 2512; // Point index invalid
					GVL.A_RunErrorStep := GVL.A_RunStep;
					GVL.A_RunState := 900;
				END_IF;
			
			
			//-------------------------------------------------------------------------
			// POINT ADD VALUE
			// P1 = Point cần thay đổi
			// P2 = X Offset
			// P3 = Y Offset
			// P4 = Z Offset
			// P5 = R Offset
			// Point[P1] := Point[P1] + Value
			//-------------------------------------------------------------------------
			E_RobotCmd.CMD_POINT_ADD_VALUE:
				IF (step_PRG_A_Interpreter.P1 >= 1) AND (step_PRG_A_Interpreter.P1 <= 500) THEN
			
					GVL_1.DATA_RB_A.X_POS[step_PRG_A_Interpreter.P1] := GVL_1.DATA_RB_A.X_POS[step_PRG_A_Interpreter.P1] + INT_TO_REAL(step_PRG_A_Interpreter.P2)/1000;
					GVL_1.DATA_RB_A.Y_POS[step_PRG_A_Interpreter.P1] := GVL_1.DATA_RB_A.Y_POS[step_PRG_A_Interpreter.P1] + DINT_TO_REAL(step_PRG_A_Interpreter.P3)/1000;
					GVL_1.DATA_RB_A.Z_POS[step_PRG_A_Interpreter.P1] := GVL_1.DATA_RB_A.Z_POS[step_PRG_A_Interpreter.P1] + INT_TO_REAL(step_PRG_A_Interpreter.P4)/1000;
					GVL_1.DATA_RB_A.R_POS[step_PRG_A_Interpreter.P1] := GVL_1.DATA_RB_A.R_POS[step_PRG_A_Interpreter.P1] + INT_TO_REAL(step_PRG_A_Interpreter.P5)/1000;
			
					GVL.A_RunStep := GVL.A_RunStep + 1;
					GVL.A_RunState := 0;
					IF GVL.A_RunMode = 1 THEN
						GVL.A_StepHold := TRUE;
					END_IF;
			
				ELSE
					GVL.A_RunAlarm := TRUE;
					GVL.A_RunAlarmCode := 2513; // Point index invalid
					GVL.A_RunErrorStep := GVL.A_RunStep;
					GVL.A_RunState := 900;
				END_IF;
			
			
			//-------------------------------------------------------------------------
			// POINT ADD INTERNAL REGISTER
			// P1 = Point cần thay đổi
			// P2 = A_Reg chứa X Offset
			// P3 = A_Reg chứa Y Offset
			// P4 = A_Reg chứa Z Offset
			// P5 = A_Reg chứa R Offset
			// Point[P1] := Point[P1] + A_Reg[]
			//-------------------------------------------------------------------------
			E_RobotCmd.CMD_POINT_ADD_REG:
				IF (step_PRG_A_Interpreter.P1 >= 1) AND (step_PRG_A_Interpreter.P1 <= 500)
				AND (step_PRG_A_Interpreter.P2 >= 1) AND (step_PRG_A_Interpreter.P2 <= 200)
				AND (step_PRG_A_Interpreter.P3 >= 1) AND (step_PRG_A_Interpreter.P3 <= 200)
				AND (step_PRG_A_Interpreter.P4 >= 1) AND (step_PRG_A_Interpreter.P4 <= 200)
				AND (step_PRG_A_Interpreter.P5 >= 1) AND (step_PRG_A_Interpreter.P5 <= 200) THEN
			
					GVL_1.DATA_RB_A.X_POS[step_PRG_A_Interpreter.P1] := GVL_1.DATA_RB_A.X_POS[step_PRG_A_Interpreter.P1] + DINT_TO_REAL(GVL.A_Reg[step_PRG_A_Interpreter.P2])/1000;
					GVL_1.DATA_RB_A.Y_POS[step_PRG_A_Interpreter.P1] := GVL_1.DATA_RB_A.Y_POS[step_PRG_A_Interpreter.P1] + DINT_TO_REAL(GVL.A_Reg[step_PRG_A_Interpreter.P3])/1000;
					GVL_1.DATA_RB_A.Z_POS[step_PRG_A_Interpreter.P1] := GVL_1.DATA_RB_A.Z_POS[step_PRG_A_Interpreter.P1] + DINT_TO_REAL(GVL.A_Reg[step_PRG_A_Interpreter.P4])/1000;
					GVL_1.DATA_RB_A.R_POS[step_PRG_A_Interpreter.P1] := GVL_1.DATA_RB_A.R_POS[step_PRG_A_Interpreter.P1] + DINT_TO_REAL(GVL.A_Reg[step_PRG_A_Interpreter.P5])/1000;
			
					GVL.A_RunStep := GVL.A_RunStep + 1;
					GVL.A_RunState := 0;
					IF GVL.A_RunMode = 1 THEN
						GVL.A_StepHold := TRUE;
					END_IF;
			
				ELSE
					GVL.A_RunAlarm := TRUE;
					GVL.A_RunAlarmCode := 2514; // Point/Reg index invalid
					GVL.A_RunErrorStep := GVL.A_RunStep;
					GVL.A_RunState := 900;
				END_IF;
			
			
			//-------------------------------------------------------------------------
			// POINT ADD MODBUS REGISTER
			// P1 = Point cần thay đổi
			// P2 = MODBUS X Offset
			// P3 = MODBUS Y Offset
			// P4 = MODBUS Z Offset
			// P5 = MODBUS R Offset
			//
			// MODBUS = 16-bit signed [-32768..32767]
			// Point[P1] := Point[P1] + MODBUS[]
			//-------------------------------------------------------------------------
			E_RobotCmd.CMD_POINT_ADD_MB_REG:
				IF (step_PRG_A_Interpreter.P1 >= 1) AND (step_PRG_A_Interpreter.P1 <= 500)
				AND (step_PRG_A_Interpreter.P2 >= 0) AND (step_PRG_A_Interpreter.P2 <= 1999)
				AND (step_PRG_A_Interpreter.P3 >= 0) AND (step_PRG_A_Interpreter.P3 <= 1999)
				AND (step_PRG_A_Interpreter.P4 >= 0) AND (step_PRG_A_Interpreter.P4 <= 1999)
				AND (step_PRG_A_Interpreter.P5 >= 0) AND (step_PRG_A_Interpreter.P5 <= 1999) THEN
			
					GVL_1.DATA_RB_A.X_POS[step_PRG_A_Interpreter.P1] := GVL_1.DATA_RB_A.X_POS[step_PRG_A_Interpreter.P1] + INT_TO_REAL(WORD_TO_INT(GVL.MODBUS[step_PRG_A_Interpreter.P2]))/1000;
					GVL_1.DATA_RB_A.Y_POS[step_PRG_A_Interpreter.P1] := GVL_1.DATA_RB_A.Y_POS[step_PRG_A_Interpreter.P1] + INT_TO_REAL(WORD_TO_INT(GVL.MODBUS[step_PRG_A_Interpreter.P3]))/1000;
					GVL_1.DATA_RB_A.Z_POS[step_PRG_A_Interpreter.P1] := GVL_1.DATA_RB_A.Z_POS[step_PRG_A_Interpreter.P1] + INT_TO_REAL(WORD_TO_INT(GVL.MODBUS[step_PRG_A_Interpreter.P4]))/1000;
					GVL_1.DATA_RB_A.R_POS[step_PRG_A_Interpreter.P1] := GVL_1.DATA_RB_A.R_POS[step_PRG_A_Interpreter.P1] + INT_TO_REAL(WORD_TO_INT(GVL.MODBUS[step_PRG_A_Interpreter.P5]))/1000;
			
					GVL.A_RunStep := GVL.A_RunStep + 1;
					GVL.A_RunState := 0;
					IF GVL.A_RunMode = 1 THEN
						GVL.A_StepHold := TRUE;
					END_IF;
			
				ELSE
					GVL.A_RunAlarm := TRUE;
					GVL.A_RunAlarmCode := 2515; // Point/MODBUS index invalid
					GVL.A_RunErrorStep := GVL.A_RunStep;
					GVL.A_RunState := 900;
				END_IF;
	
				
			E_RobotCmd.CMD_REG_SET,
			E_RobotCmd.CMD_REG_ADD,
			E_RobotCmd.CMD_REG_SUB,
			E_RobotCmd.CMD_REG_MUL,
			E_RobotCmd.CMD_REG_DIV,
			E_RobotCmd.CMD_REG_MOD:
			
				// P1 = Reg đích
				// P2 = SourceMode
				// P3 = Value hoặc Reg A
				// P4 = Reg B
			
				IF (step_PRG_A_Interpreter.P1 >= 1) AND (step_PRG_A_Interpreter.P1 <= 200) THEN
			
					GVL.A_Reg[step_PRG_A_Interpreter.P1] :=
						F_CalcReg_A(
							Cmd        := step_PRG_A_Interpreter.Cmd,
							DestReg    := step_PRG_A_Interpreter.P1,
							SourceMode := step_PRG_A_Interpreter.P2,
							P3         := step_PRG_A_Interpreter.P3,
							P4         := step_PRG_A_Interpreter.P4
						);
			
					GVL.A_RunStep := GVL.A_RunStep + 1;
					GVL.A_RunState := 0;
					// Nếu đang Step Mode thì dừng chờ sau khi chạy xong 1 lệnh
					IF GVL.A_RunMode = 1 THEN
						GVL.A_StepHold := TRUE;
					END_IF;
			
				ELSE
					GVL.A_RunAlarm := TRUE;
					GVL.A_RunAlarmCode := 2401; // Reg index invalid
					GVL.A_RunErrorStep := GVL.A_RunStep;
					GVL.A_RunState := 900;
				END_IF;
				
				
			E_RobotCmd.CMD_VAR_SET,
			E_RobotCmd.CMD_VAR_ADD,
			E_RobotCmd.CMD_VAR_SUB,
			E_RobotCmd.CMD_VAR_MUL,
			E_RobotCmd.CMD_VAR_DIV,
			E_RobotCmd.CMD_VAR_MOD:
				// P1 = Var đích
				// P2 = SourceMode
				// P3 = Value hoặc Var A
				// P4 = Var B
				IF (step_PRG_A_Interpreter.P1 >= 1) AND (step_PRG_A_Interpreter.P1 <= 200) THEN
			
					GVL.A_Var[step_PRG_A_Interpreter.P1] :=
						F_CalcVar_A(
							Cmd        := step_PRG_A_Interpreter.Cmd,
							DestVar    := step_PRG_A_Interpreter.P1,
							SourceMode := step_PRG_A_Interpreter.P2,
							P3         := step_PRG_A_Interpreter.P3,
							P4         := step_PRG_A_Interpreter.P4
						);
			
					GVL.A_RunStep := GVL.A_RunStep + 1;
					GVL.A_RunState := 0;
					// Nếu đang Step Mode thì dừng chờ sau khi chạy xong 1 lệnh
					IF GVL.A_RunMode = 1 THEN
						GVL.A_StepHold := TRUE;
					END_IF;
			
				ELSE
					GVL.A_RunAlarm := TRUE;
					GVL.A_RunAlarmCode := 2402;
					GVL.A_RunErrorStep := GVL.A_RunStep;
					GVL.A_RunState := 900;
				END_IF;
				
				
            E_RobotCmd.CMD_END:
                GVL.A_RunBusy := FALSE;
                GVL.A_RunDone := TRUE;
                GVL.A_RunState := 0;
		

        ELSE
            // Lệnh chưa hỗ trợ
            GVL.A_RunAlarm := TRUE;
            GVL.A_RunAlarmCode := 2001;
            GVL.A_RunErrorStep := GVL.A_RunStep;
            GVL.A_RunState := 900;
        END_CASE;


    100: // FILL PIPELINE

        // Nạp trước motion nếu:
        // 1. Chưa hết chương trình
        // 2. Step tiếp theo vẫn là motion
        // 3. Tổng số motion đang chờ + đang chạy chưa vượt pipeline depth
        IF (GVL.A_PipelineNextPushStep <= GVL.A_LengthStep)
           AND F_IsMotionCmd(GVL_1.Step_Cr_A[GVL.A_PipelineNextPushStep].Cmd)
           AND ((GVL.A_MotionCount + GVL.A_ActiveMotionCount) < GVL.A_PipelineDepth)
		   // AND (GVL.A_PipelineUsedCount < GVL.A_PipelineDepth)
        THEN
            GVL.A_PushMotionItem := F_BuildMotionItem(GVL.A_PipelineNextPushStep);
            GVL.A_PushMotionReq := TRUE;

            GVL.A_RunState := 110;
        ELSE
            // Pipeline đã đầy hoặc gặp lệnh logic
            GVL.A_RunState := 120;
        END_IF;


    110: // WAIT PUSH DONE
		
			IF GVL.A_PushMotionDone THEN
			
					GVL.A_PushMotionReq := FALSE;
					GVL.A_PushMotionDone := FALSE;
					
					//------------------------------------------------
					// Một motion chính thức thuộc pipeline
					//------------------------------------------------
					GVL.A_PipelineUsedCount :=
						GVL.A_PipelineUsedCount + 1;
			
					GVL.A_PipelineNextPushStep :=
						GVL.A_PipelineNextPushStep + 1;

					// Chờ motion hiện tại hoàn thành
					//GVL.A_RunState := 120;
					//GVL.A_RunState := 100;
					//------------------------------------------------
					// Kiểm tra BlendMode của Motion hiện tại
					//
					// P3:
					// 0  = Không Blending
					// >0 = Có Blending
					//------------------------------------------------
					
					IF GVL.A_RunMode = 0 THEN
						//IF (GVL_1.Step_Cr_A[GVL.A_PipelineNextPushStep - 1].P3 > 0) AND (GVL_1.Step_Cr_A[GVL.A_PipelineNextPushStep].P3 > 0) THEN
						IF (GVL_1.Step_Cr_A[GVL.A_PipelineNextPushStep - 1].P3 > 0) THEN
							//--------------------------------------------
							// Có Blending:
							// quay lại State100 để preload Motion tiếp
							//--------------------------------------------
							GVL.A_RunState := 100;
				
						ELSE
				
							//--------------------------------------------
							// Không Blending:
							// không preload tiếp.
							// Chờ Motion hiện tại Done + Check Position.
							//--------------------------------------------
							//GVL.A_RunState := 120;
							GVL.A_RunState := 100;
				
						END_IF;
					ELSE
						GVL.A_RunState := 120;
					END_IF;
			
			
				ELSIF GVL.A_PushMotionError THEN
			
					GVL.A_PushMotionReq := FALSE;
			
					GVL.A_RunAlarm := TRUE;
					GVL.A_RunAlarmCode := 3001;
					GVL.A_RunErrorStep :=
						GVL.A_PipelineNextPushStep;
			
					GVL.A_RunState := 900;
			
				END_IF;

    120: // WAIT CURRENT STEP DONE
		IF GVL.A_MotionErrorPulse THEN

			GVL.A_RunAlarm := TRUE;
			GVL.A_RunErrorStep := GVL.A_MotionErrorStep;
			GVL.A_RunAlarmCode := GVL.A_MotionErrorCode;
	
			GVL.A_MotionErrorPulse := FALSE;
			GVL.A_RunState := 900;
	
	
		ELSIF GVL.A_MotionDonePulse
			  AND (GVL.A_MotionDoneStep = GVL.A_RunStep)
		THEN
	
			//--------------------------------------------
			// Tiêu thụ Done của step hiện tại
			//--------------------------------------------
			GVL.A_MotionDonePulse := FALSE;
			GVL.A_MotionDoneStep := 0;
	
			//--------------------------------------------
			// Sang step tiếp theo
			//--------------------------------------------
			GVL.A_RunStep :=
				GVL.A_RunStep + 1;
	
